REGION Network 58: Falownik P3
   // Sterowaniem pracy z falownika. Sterowanie napędem na pozycji MC
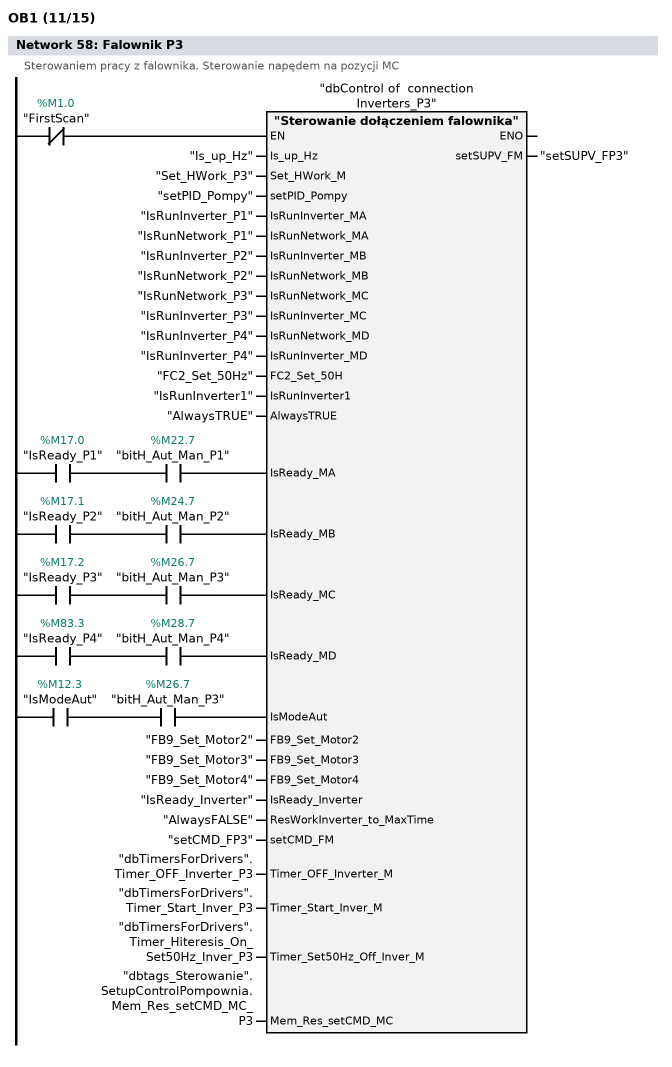
   RUNG wire#powerrail
      I_Contact( "FirstScan" )
      "dbControl of  connection Inverters_P3"(IsReady_MA := wire#w1, IsReady_MB := wire#w2, IsReady_MC := wire#w3, IsReady_MD := wire#w4, IsModeAut := wire#w5, Is_up_Hz := "Is_up_Hz", Set_HWork_M := "Set_HWork_P3", setPID_Pompy := "setPID_Pompy", IsRunInverter_MA := "IsRunInverter_P1", IsRunNetwork_MA := "IsRunNetwork_P1", IsRunInverter_MB := "IsRunInverter_P2", IsRunNetwork_MB := "IsRunNetwork_P2", IsRunNetwork_MC := "IsRunNetwork_P3", IsRunInverter_MC := "IsRunInverter_P3", IsRunNetwork_MD := "IsRunInverter_P4", IsRunInverter_MD := "IsRunInverter_P4", FC2_Set_50H := "FC2_Set_50Hz", IsRunInverter1 := "IsRunInverter1", AlwaysTRUE := "AlwaysTRUE", FB9_Set_Motor2 := "FB9_Set_Motor2", FB9_Set_Motor3 := "FB9_Set_Motor3", FB9_Set_Motor4 := "FB9_Set_Motor4", IsReady_Inverter := "IsReady_Inverter", ResWorkInverter_to_MaxTime := "AlwaysFALSE", setCMD_FM := "setCMD_FP3", Timer_OFF_Inverter_M := "dbTimersForDrivers".Timer_OFF_Inverter_P3, Timer_Start_Inver_M := "dbTimersForDrivers".Timer_Start_Inver_P3, Timer_Set50Hz_Off_Inver_M := "dbTimersForDrivers".Timer_Hiteresis_On_Set50Hz_Inver_P3, Mem_Res_setCMD_MC := "dbtags_Sterowanie".SetupControlPompownia.Mem_Res_setCMD_MC_P3, setSUPV_FM => "setSUPV_FP3")
   END_RUNG
   RUNG wire#powerrail
      Contact( "IsReady_P1" )
      Contact( "bitH_Aut_Man_P1" )
   END_RUNG wire#w1
   RUNG wire#powerrail
      Contact( "IsReady_P2" )
      Contact( "bitH_Aut_Man_P2" )
   END_RUNG wire#w2
   RUNG wire#powerrail
      Contact( "IsReady_P3" )
      Contact( "bitH_Aut_Man_P3" )
   END_RUNG wire#w3
   RUNG wire#powerrail
      Contact( "IsReady_P4" )
      Contact( "bitH_Aut_Man_P4" )
   END_RUNG wire#w4
   RUNG wire#powerrail
      Contact( "IsModeAut" )
      Contact( "bitH_Aut_Man_P3" )
   END_RUNG wire#w5
   // the same network as SCL:
   IF NOT "FirstScan" THEN
       "dbControl of  connection Inverters_P3"(Is_up_Hz := "Is_up_Hz",   // "Sterowanie dołączeniem falownika"
                               Set_HWork_M := "Set_HWork_P3",
                               setPID_Pompy := "setPID_Pompy",
                               IsRunInverter_MA := "IsRunInverter_P1",
                               IsRunNetwork_MA := "IsRunNetwork_P1",
                               IsRunInverter_MB := "IsRunInverter_P2",
                               IsRunNetwork_MB := "IsRunNetwork_P2",
                               IsRunNetwork_MC := "IsRunNetwork_P3",
                               IsRunInverter_MC := "IsRunInverter_P3",
                               IsRunNetwork_MD := "IsRunInverter_P4",
                               IsRunInverter_MD := "IsRunInverter_P4",
                               FC2_Set_50H := "FC2_Set_50Hz",
                               IsRunInverter1 := "IsRunInverter1",
                               AlwaysTRUE := "AlwaysTRUE",
                               IsReady_MA := "IsReady_P1" AND "bitH_Aut_Man_P1",
                               IsReady_MB := "IsReady_P2" AND "bitH_Aut_Man_P2",
                               IsReady_MC := "IsReady_P3" AND "bitH_Aut_Man_P3",
                               IsReady_MD := "IsReady_P4" AND "bitH_Aut_Man_P4",
                               IsModeAut := "IsModeAut" AND "bitH_Aut_Man_P3",
                               FB9_Set_Motor2 := "FB9_Set_Motor2",
                               FB9_Set_Motor3 := "FB9_Set_Motor3",
                               FB9_Set_Motor4 := "FB9_Set_Motor4",
                               IsReady_Inverter := "IsReady_Inverter",
                               ResWorkInverter_to_MaxTime := "AlwaysFALSE",
                               setCMD_FM := "setCMD_FP3",
                               Timer_OFF_Inverter_M := "dbTimersForDrivers".Timer_OFF_Inverter_P3,
                               Timer_Start_Inver_M := "dbTimersForDrivers".Timer_Start_Inver_P3,
                               Timer_Set50Hz_Off_Inver_M := "dbTimersForDrivers".Timer_Hiteresis_On_Set50Hz_Inver_P3,
                               Mem_Res_setCMD_MC := "dbtags_Sterowanie".SetupControlPompownia.Mem_Res_setCMD_MC_P3,
                               setSUPV_FM => "setSUPV_FP3");
   END_IF;
END_REGION

REGION Network 59: Falownik P4
   // Sterowaniem pracy z falownika. Sterowanie napędem na pozycji MC
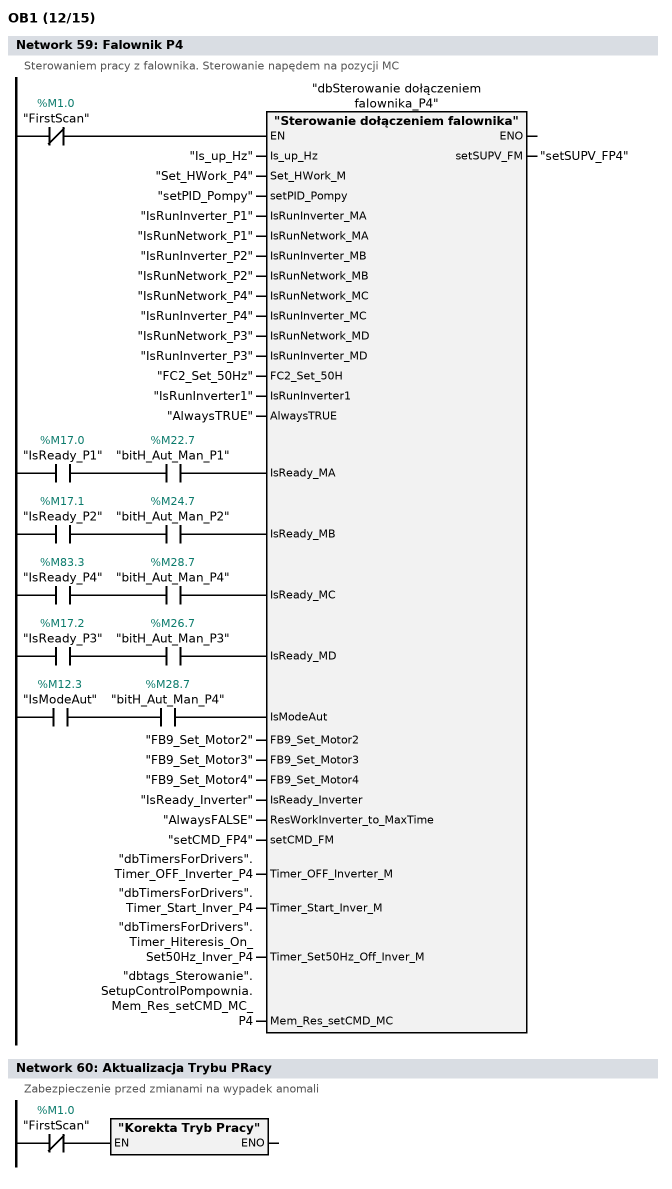
   RUNG wire#powerrail
      I_Contact( "FirstScan" )
      "dbSterowanie dołączeniem falownika_P4"(IsReady_MA := wire#w1, IsReady_MB := wire#w2, IsReady_MC := wire#w3, IsReady_MD := wire#w4, IsModeAut := wire#w5, Is_up_Hz := "Is_up_Hz", Set_HWork_M := "Set_HWork_P4", setPID_Pompy := "setPID_Pompy", IsRunInverter_MA := "IsRunInverter_P1", IsRunNetwork_MA := "IsRunNetwork_P1", IsRunInverter_MB := "IsRunInverter_P2", IsRunNetwork_MB := "IsRunNetwork_P2", IsRunNetwork_MC := "IsRunNetwork_P4", IsRunInverter_MC := "IsRunInverter_P4", IsRunNetwork_MD := "IsRunNetwork_P3", IsRunInverter_MD := "IsRunInverter_P3", FC2_Set_50H := "FC2_Set_50Hz", IsRunInverter1 := "IsRunInverter1", AlwaysTRUE := "AlwaysTRUE", FB9_Set_Motor2 := "FB9_Set_Motor2", FB9_Set_Motor3 := "FB9_Set_Motor3", FB9_Set_Motor4 := "FB9_Set_Motor4", IsReady_Inverter := "IsReady_Inverter", ResWorkInverter_to_MaxTime := "AlwaysFALSE", setCMD_FM := "setCMD_FP4", Timer_OFF_Inverter_M := "dbTimersForDrivers".Timer_OFF_Inverter_P4, Timer_Start_Inver_M := "dbTimersForDrivers".Timer_Start_Inver_P4, Timer_Set50Hz_Off_Inver_M := "dbTimersForDrivers".Timer_Hiteresis_On_Set50Hz_Inver_P4, Mem_Res_setCMD_MC := "dbtags_Sterowanie".SetupControlPompownia.Mem_Res_setCMD_MC_P4, setSUPV_FM => "setSUPV_FP4")
   END_RUNG
   RUNG wire#powerrail
      Contact( "IsReady_P1" )
      Contact( "bitH_Aut_Man_P1" )
   END_RUNG wire#w1
   RUNG wire#powerrail
      Contact( "IsReady_P2" )
      Contact( "bitH_Aut_Man_P2" )
   END_RUNG wire#w2
   RUNG wire#powerrail
      Contact( "IsReady_P4" )
      Contact( "bitH_Aut_Man_P4" )
   END_RUNG wire#w3
   RUNG wire#powerrail
      Contact( "IsReady_P3" )
      Contact( "bitH_Aut_Man_P3" )
   END_RUNG wire#w4
   RUNG wire#powerrail
      Contact( "IsModeAut" )
      Contact( "bitH_Aut_Man_P4" )
   END_RUNG wire#w5
   // the same network as SCL:
   IF NOT "FirstScan" THEN
       "dbSterowanie dołączeniem falownika_P4"(Is_up_Hz := "Is_up_Hz",   // "Sterowanie dołączeniem falownika"
                               Set_HWork_M := "Set_HWork_P4",
                               setPID_Pompy := "setPID_Pompy",
                               IsRunInverter_MA := "IsRunInverter_P1",
                               IsRunNetwork_MA := "IsRunNetwork_P1",
                               IsRunInverter_MB := "IsRunInverter_P2",
                               IsRunNetwork_MB := "IsRunNetwork_P2",
                               IsRunNetwork_MC := "IsRunNetwork_P4",
                               IsRunInverter_MC := "IsRunInverter_P4",
                               IsRunNetwork_MD := "IsRunNetwork_P3",
                               IsRunInverter_MD := "IsRunInverter_P3",
                               FC2_Set_50H := "FC2_Set_50Hz",
                               IsRunInverter1 := "IsRunInverter1",
                               AlwaysTRUE := "AlwaysTRUE",
                               IsReady_MA := "IsReady_P1" AND "bitH_Aut_Man_P1",
                               IsReady_MB := "IsReady_P2" AND "bitH_Aut_Man_P2",
                               IsReady_MC := "IsReady_P4" AND "bitH_Aut_Man_P4",
                               IsReady_MD := "IsReady_P3" AND "bitH_Aut_Man_P3",
                               IsModeAut := "IsModeAut" AND "bitH_Aut_Man_P4",
                               FB9_Set_Motor2 := "FB9_Set_Motor2",
                               FB9_Set_Motor3 := "FB9_Set_Motor3",
                               FB9_Set_Motor4 := "FB9_Set_Motor4",
                               IsReady_Inverter := "IsReady_Inverter",
                               ResWorkInverter_to_MaxTime := "AlwaysFALSE",
                               setCMD_FM := "setCMD_FP4",
                               Timer_OFF_Inverter_M := "dbTimersForDrivers".Timer_OFF_Inverter_P4,
                               Timer_Start_Inver_M := "dbTimersForDrivers".Timer_Start_Inver_P4,
                               Timer_Set50Hz_Off_Inver_M := "dbTimersForDrivers".Timer_Hiteresis_On_Set50Hz_Inver_P4,
                               Mem_Res_setCMD_MC := "dbtags_Sterowanie".SetupControlPompownia.Mem_Res_setCMD_MC_P4,
                               setSUPV_FM => "setSUPV_FP4");
   END_IF;
END_REGION

REGION Network 60: Aktualizacja Trybu PRacy
   // Zabezpieczenie przed zmianami na wypadek anomali
   RUNG wire#powerrail
      I_Contact( "FirstScan" )
      "Korekta Tryb Pracy"()
   END_RUNG
   // the same network as SCL:
   IF NOT "FirstScan" THEN "Korekta Tryb Pracy"(); END_IF;
END_REGION

REGION Network 61: Sterowanie falownikiem
   // Sterowanie załaczaniem falownika
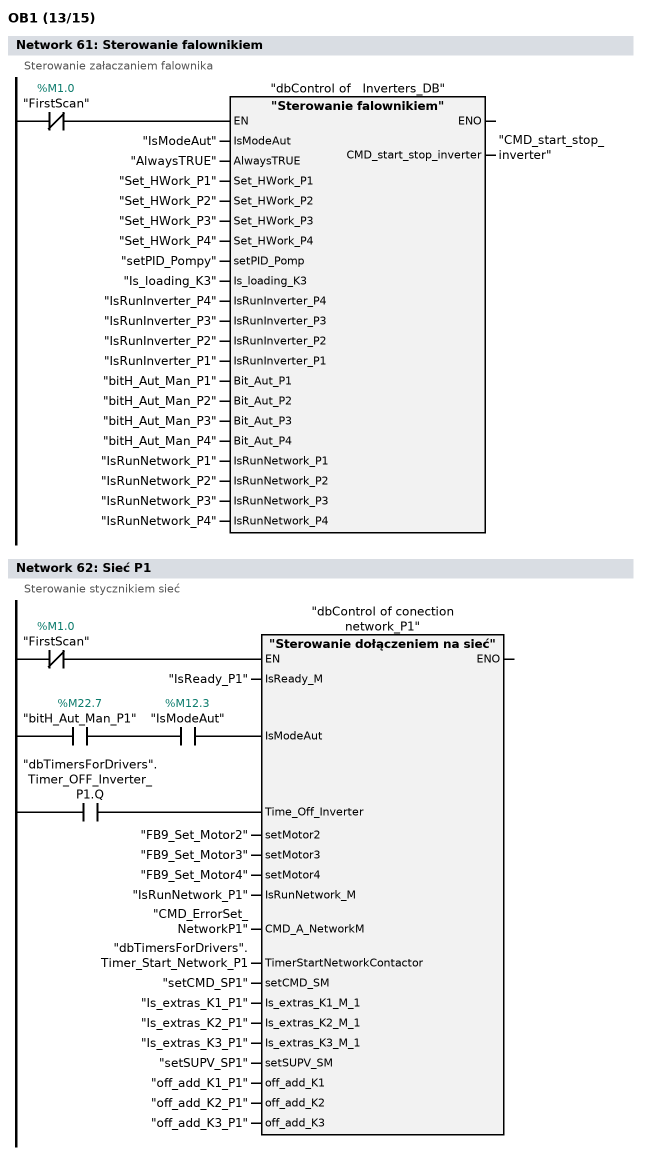
   RUNG wire#powerrail
      I_Contact( "FirstScan" )
      "dbControl of   Inverters_DB"(IsModeAut := "IsModeAut", AlwaysTRUE := "AlwaysTRUE", Set_HWork_P1 := "Set_HWork_P1", Set_HWork_P2 := "Set_HWork_P2", Set_HWork_P3 := "Set_HWork_P3", Set_HWork_P4 := "Set_HWork_P4", setPID_Pomp := "setPID_Pompy", Is_loading_K3 := "Is_loading_K3", IsRunInverter_P4 := "IsRunInverter_P4", IsRunInverter_P3 := "IsRunInverter_P3", IsRunInverter_P2 := "IsRunInverter_P2", IsRunInverter_P1 := "IsRunInverter_P1", Bit_Aut_P1 := "bitH_Aut_Man_P1", Bit_Aut_P2 := "bitH_Aut_Man_P2", Bit_Aut_P3 := "bitH_Aut_Man_P3", Bit_Aut_P4 := "bitH_Aut_Man_P4", IsRunNetwork_P1 := "IsRunNetwork_P1", IsRunNetwork_P2 := "IsRunNetwork_P2", IsRunNetwork_P3 := "IsRunNetwork_P3", IsRunNetwork_P4 := "IsRunNetwork_P4", CMD_start_stop_inverter => "CMD_start_stop_inverter")
   END_RUNG
   // the same network as SCL:
   IF NOT "FirstScan" THEN
       "dbControl of   Inverters_DB"(IsModeAut := "IsModeAut",   // "Sterowanie falownikiem"
                               AlwaysTRUE := "AlwaysTRUE",
                               Set_HWork_P1 := "Set_HWork_P1",
                               Set_HWork_P2 := "Set_HWork_P2",
                               Set_HWork_P3 := "Set_HWork_P3",
                               Set_HWork_P4 := "Set_HWork_P4",
                               setPID_Pomp := "setPID_Pompy",
                               Is_loading_K3 := "Is_loading_K3",
                               IsRunInverter_P4 := "IsRunInverter_P4",
                               IsRunInverter_P3 := "IsRunInverter_P3",
                               IsRunInverter_P2 := "IsRunInverter_P2",
                               IsRunInverter_P1 := "IsRunInverter_P1",
                               Bit_Aut_P1 := "bitH_Aut_Man_P1",
                               Bit_Aut_P2 := "bitH_Aut_Man_P2",
                               Bit_Aut_P3 := "bitH_Aut_Man_P3",
                               Bit_Aut_P4 := "bitH_Aut_Man_P4",
                               IsRunNetwork_P1 := "IsRunNetwork_P1",
                               IsRunNetwork_P2 := "IsRunNetwork_P2",
                               IsRunNetwork_P3 := "IsRunNetwork_P3",
                               IsRunNetwork_P4 := "IsRunNetwork_P4",
                               CMD_start_stop_inverter => "CMD_start_stop_inverter");
   END_IF;
END_REGION

REGION Network 62: Sieć P1
   // Sterowanie stycznikiem sieć
   RUNG wire#powerrail
      I_Contact( "FirstScan" )
      "dbControl of conection network_P1"(IsModeAut := wire#w1, Time_Off_Inverter := wire#w2, IsReady_M := "IsReady_P1", setMotor2 := "FB9_Set_Motor2", setMotor3 := "FB9_Set_Motor3", setMotor4 := "FB9_Set_Motor4", IsRunNetwork_M := "IsRunNetwork_P1", CMD_A_NetworkM := "CMD_ErrorSet_NetworkP1", TimerStartNetworkContactor := "dbTimersForDrivers".Timer_Start_Network_P1, setCMD_SM := "setCMD_SP1", Is_extras_K1_M_1 := "Is_extras_K1_P1", Is_extras_K2_M_1 := "Is_extras_K2_P1", Is_extras_K3_M_1 := "Is_extras_K3_P1", setSUPV_SM := "setSUPV_SP1", off_add_K1 := "off_add_K1_P1", off_add_K2 := "off_add_K2_P1", off_add_K3 := "off_add_K3_P1")
   END_RUNG
   RUNG wire#powerrail
      Contact( "bitH_Aut_Man_P1" )
      Contact( "IsModeAut" )
   END_RUNG wire#w1
   RUNG wire#powerrail
      Contact( "dbTimersForDrivers".Timer_OFF_Inverter_P1.Q )
   END_RUNG wire#w2
   // the same network as SCL:
   IF NOT "FirstScan" THEN
       "dbControl of conection network_P1"(IsReady_M := "IsReady_P1",   // "Sterowanie dołączeniem na sieć"
                               IsModeAut := "bitH_Aut_Man_P1" AND "IsModeAut",
                               Time_Off_Inverter := "dbTimersForDrivers".Timer_OFF_Inverter_P1.Q,
                               setMotor2 := "FB9_Set_Motor2",
                               setMotor3 := "FB9_Set_Motor3",
                               setMotor4 := "FB9_Set_Motor4",
                               IsRunNetwork_M := "IsRunNetwork_P1",
                               CMD_A_NetworkM := "CMD_ErrorSet_NetworkP1",
                               TimerStartNetworkContactor := "dbTimersForDrivers".Timer_Start_Network_P1,
                               setCMD_SM := "setCMD_SP1",
                               Is_extras_K1_M_1 := "Is_extras_K1_P1",
                               Is_extras_K2_M_1 := "Is_extras_K2_P1",
                               Is_extras_K3_M_1 := "Is_extras_K3_P1",
                               setSUPV_SM := "setSUPV_SP1",
                               off_add_K1 := "off_add_K1_P1",
                               off_add_K2 := "off_add_K2_P1",
                               off_add_K3 := "off_add_K3_P1");
   END_IF;
END_REGION

REGION Network 63: Sieć P2
   // Sterowanie stycznikiem sieć
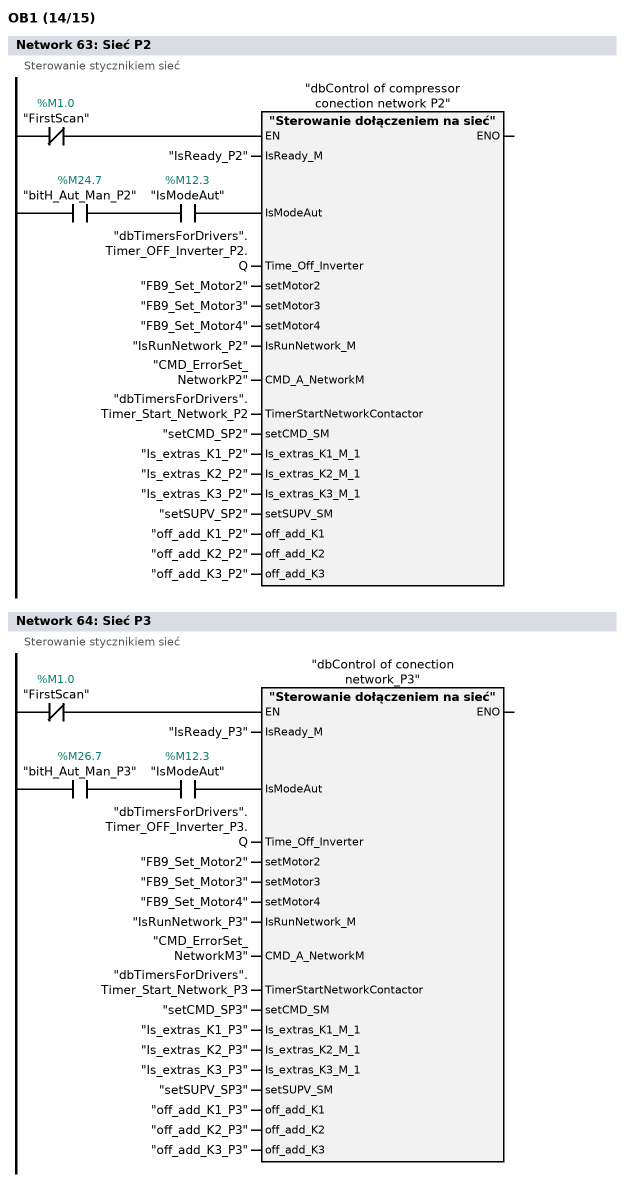
   RUNG wire#powerrail
      I_Contact( "FirstScan" )
      "dbControl of compressor conection network P2"(IsModeAut := wire#w1, IsReady_M := "IsReady_P2", Time_Off_Inverter := "dbTimersForDrivers".Timer_OFF_Inverter_P2.Q, setMotor2 := "FB9_Set_Motor2", setMotor3 := "FB9_Set_Motor3", setMotor4 := "FB9_Set_Motor4", IsRunNetwork_M := "IsRunNetwork_P2", CMD_A_NetworkM := "CMD_ErrorSet_NetworkP2", TimerStartNetworkContactor := "dbTimersForDrivers".Timer_Start_Network_P2, setCMD_SM := "setCMD_SP2", Is_extras_K1_M_1 := "Is_extras_K1_P2", Is_extras_K2_M_1 := "Is_extras_K2_P2", Is_extras_K3_M_1 := "Is_extras_K3_P2", setSUPV_SM := "setSUPV_SP2", off_add_K1 := "off_add_K1_P2", off_add_K2 := "off_add_K2_P2", off_add_K3 := "off_add_K3_P2")
   END_RUNG
   RUNG wire#powerrail
      Contact( "bitH_Aut_Man_P2" )
      Contact( "IsModeAut" )
   END_RUNG wire#w1
   // the same network as SCL:
   IF NOT "FirstScan" THEN
       "dbControl of compressor conection network P2"(IsReady_M := "IsReady_P2",   // "Sterowanie dołączeniem na sieć"
                               IsModeAut := "bitH_Aut_Man_P2" AND "IsModeAut",
                               Time_Off_Inverter := "dbTimersForDrivers".Timer_OFF_Inverter_P2.Q,
                               setMotor2 := "FB9_Set_Motor2",
                               setMotor3 := "FB9_Set_Motor3",
                               setMotor4 := "FB9_Set_Motor4",
                               IsRunNetwork_M := "IsRunNetwork_P2",
                               CMD_A_NetworkM := "CMD_ErrorSet_NetworkP2",
                               TimerStartNetworkContactor := "dbTimersForDrivers".Timer_Start_Network_P2,
                               setCMD_SM := "setCMD_SP2",
                               Is_extras_K1_M_1 := "Is_extras_K1_P2",
                               Is_extras_K2_M_1 := "Is_extras_K2_P2",
                               Is_extras_K3_M_1 := "Is_extras_K3_P2",
                               setSUPV_SM := "setSUPV_SP2",
                               off_add_K1 := "off_add_K1_P2",
                               off_add_K2 := "off_add_K2_P2",
                               off_add_K3 := "off_add_K3_P2");
   END_IF;
END_REGION

REGION Network 64: Sieć P3
   // Sterowanie stycznikiem sieć
   RUNG wire#powerrail
      I_Contact( "FirstScan" )
      "dbControl of conection network_P3"(IsModeAut := wire#w1, IsReady_M := "IsReady_P3", Time_Off_Inverter := "dbTimersForDrivers".Timer_OFF_Inverter_P3.Q, setMotor2 := "FB9_Set_Motor2", setMotor3 := "FB9_Set_Motor3", setMotor4 := "FB9_Set_Motor4", IsRunNetwork_M := "IsRunNetwork_P3", CMD_A_NetworkM := "CMD_ErrorSet_NetworkM3", TimerStartNetworkContactor := "dbTimersForDrivers".Timer_Start_Network_P3, setCMD_SM := "setCMD_SP3", Is_extras_K1_M_1 := "Is_extras_K1_P3", Is_extras_K2_M_1 := "Is_extras_K2_P3", Is_extras_K3_M_1 := "Is_extras_K3_P3", setSUPV_SM := "setSUPV_SP3", off_add_K1 := "off_add_K1_P3", off_add_K2 := "off_add_K2_P3", off_add_K3 := "off_add_K3_P3")
   END_RUNG
   RUNG wire#powerrail
      Contact( "bitH_Aut_Man_P3" )
      Contact( "IsModeAut" )
   END_RUNG wire#w1
   // the same network as SCL:
   IF NOT "FirstScan" THEN
       "dbControl of conection network_P3"(IsReady_M := "IsReady_P3",   // "Sterowanie dołączeniem na sieć"
                               IsModeAut := "bitH_Aut_Man_P3" AND "IsModeAut",
                               Time_Off_Inverter := "dbTimersForDrivers".Timer_OFF_Inverter_P3.Q,
                               setMotor2 := "FB9_Set_Motor2",
                               setMotor3 := "FB9_Set_Motor3",
                               setMotor4 := "FB9_Set_Motor4",
                               IsRunNetwork_M := "IsRunNetwork_P3",
                               CMD_A_NetworkM := "CMD_ErrorSet_NetworkM3",
                               TimerStartNetworkContactor := "dbTimersForDrivers".Timer_Start_Network_P3,
                               setCMD_SM := "setCMD_SP3",
                               Is_extras_K1_M_1 := "Is_extras_K1_P3",
                               Is_extras_K2_M_1 := "Is_extras_K2_P3",
                               Is_extras_K3_M_1 := "Is_extras_K3_P3",
                               setSUPV_SM := "setSUPV_SP3",
                               off_add_K1 := "off_add_K1_P3",
                               off_add_K2 := "off_add_K2_P3",
                               off_add_K3 := "off_add_K3_P3");
   END_IF;
END_REGION

REGION Network 65: Sieć P4
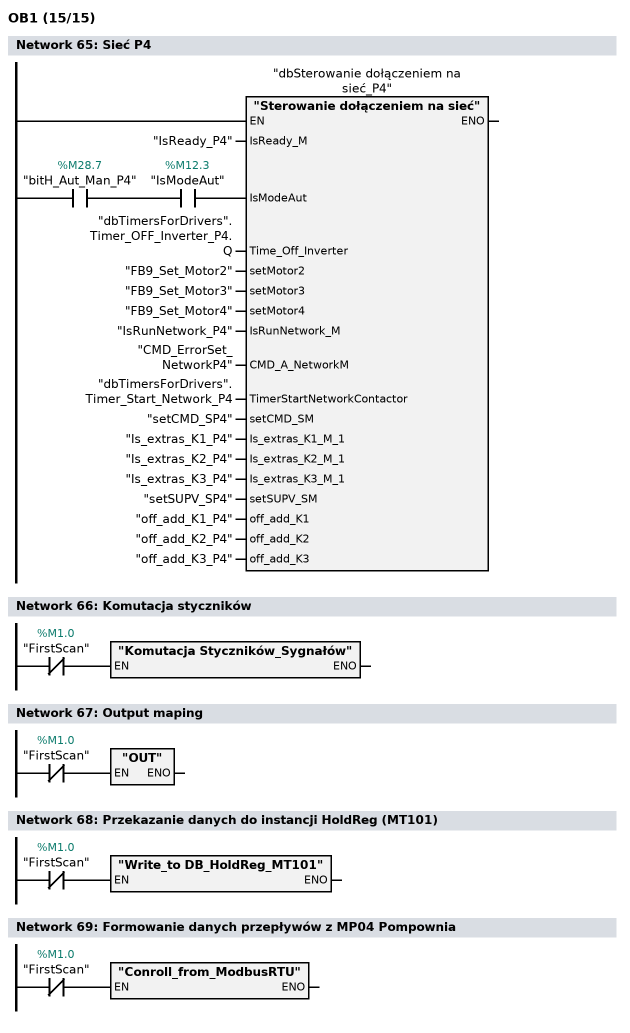
   RUNG wire#powerrail
      "dbSterowanie dołączeniem na sieć_P4"(IsModeAut := wire#w1, IsReady_M := "IsReady_P4", Time_Off_Inverter := "dbTimersForDrivers".Timer_OFF_Inverter_P4.Q, setMotor2 := "FB9_Set_Motor2", setMotor3 := "FB9_Set_Motor3", setMotor4 := "FB9_Set_Motor4", IsRunNetwork_M := "IsRunNetwork_P4", CMD_A_NetworkM := "CMD_ErrorSet_NetworkP4", TimerStartNetworkContactor := "dbTimersForDrivers".Timer_Start_Network_P4, setCMD_SM := "setCMD_SP4", Is_extras_K1_M_1 := "Is_extras_K1_P4", Is_extras_K2_M_1 := "Is_extras_K2_P4", Is_extras_K3_M_1 := "Is_extras_K3_P4", setSUPV_SM := "setSUPV_SP4", off_add_K1 := "off_add_K1_P4", off_add_K2 := "off_add_K2_P4", off_add_K3 := "off_add_K3_P4")
   END_RUNG
   RUNG wire#powerrail
      Contact( "bitH_Aut_Man_P4" )
      Contact( "IsModeAut" )
   END_RUNG wire#w1
   // the same network as SCL:
   "dbSterowanie dołączeniem na sieć_P4"(IsReady_M := "IsReady_P4",   // "Sterowanie dołączeniem na sieć"
                           IsModeAut := "bitH_Aut_Man_P4" AND "IsModeAut",
                           Time_Off_Inverter := "dbTimersForDrivers".Timer_OFF_Inverter_P4.Q,
                           setMotor2 := "FB9_Set_Motor2",
                           setMotor3 := "FB9_Set_Motor3",
                           setMotor4 := "FB9_Set_Motor4",
                           IsRunNetwork_M := "IsRunNetwork_P4",
                           CMD_A_NetworkM := "CMD_ErrorSet_NetworkP4",
                           TimerStartNetworkContactor := "dbTimersForDrivers".Timer_Start_Network_P4,
                           setCMD_SM := "setCMD_SP4",
                           Is_extras_K1_M_1 := "Is_extras_K1_P4",
                           Is_extras_K2_M_1 := "Is_extras_K2_P4",
                           Is_extras_K3_M_1 := "Is_extras_K3_P4",
                           setSUPV_SM := "setSUPV_SP4",
                           off_add_K1 := "off_add_K1_P4",
                           off_add_K2 := "off_add_K2_P4",
                           off_add_K3 := "off_add_K3_P4");
END_REGION

REGION Network 66: Komutacja styczników
   RUNG wire#powerrail
      I_Contact( "FirstScan" )
      "Komutacja Styczników_Sygnałów"()
   END_RUNG
   // the same network as SCL:
   IF NOT "FirstScan" THEN "Komutacja Styczników_Sygnałów"(); END_IF;
END_REGION

REGION Network 67: Output maping
   RUNG wire#powerrail
      I_Contact( "FirstScan" )
      "OUT"()
   END_RUNG
   // the same network as SCL:
   IF NOT "FirstScan" THEN "OUT"(); END_IF;
END_REGION

REGION Network 68: Przekazanie danych do instancji HoldReg (MT101)
   RUNG wire#powerrail
      I_Contact( "FirstScan" )
      "Write_to DB_HoldReg_MT101"()
   END_RUNG
   // the same network as SCL:
   IF NOT "FirstScan" THEN "Write_to DB_HoldReg_MT101"(); END_IF;
END_REGION

REGION Network 69: Formowanie danych przepływów z MP04 Pompownia
   RUNG wire#powerrail
      I_Contact( "FirstScan" )
      "Conroll_from_ModbusRTU"()
   END_RUNG
   // the same network as SCL:
   IF NOT "FirstScan" THEN "Conroll_from_ModbusRTU"(); END_IF;
END_REGION
END_ORGANIZATION_BLOCK

FUNCTION "RTC" : Void   // FC44, LAD
{ S7_Optimized_Access := 'TRUE' }
VERSION : 0.1
// stored: AutoNumber true, IsIECCheckEnabled false, SetENOAutomatically false, UDAEnableTagReadback false
   VAR_TEMP   // added for the SCL form of the ladder/FBD networks
      _w1 : Bool;
      _w2 : Bool;
   END_VAR
BEGIN

REGION Network 1
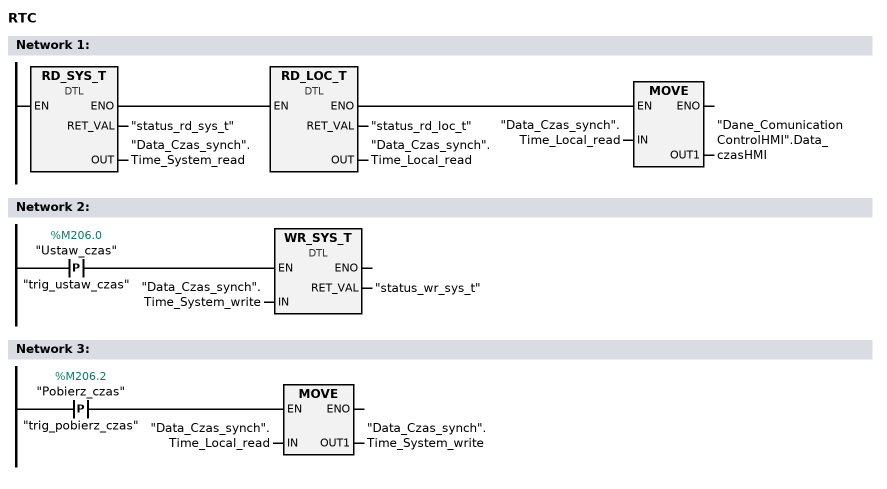
   RUNG wire#powerrail
      { S7_Templates := "date_type := DTL" } RD_SYS_T(RET_VAL => "status_rd_sys_t", OUT => "Data_Czas_synch".Time_System_read)
      { S7_Templates := "date_type := DTL" } RD_LOC_T(RET_VAL => "status_rd_loc_t", OUT => "Data_Czas_synch".Time_Local_read)
      { S7_GenerateENO := "TRUE" } Move(in := "Data_Czas_synch".Time_Local_read, out1 => "Dane_ComunicationControlHMI".Data_czasHMI)
   END_RUNG
   // the same network as SCL:
   "status_rd_sys_t" := RD_SYS_T(OUT => "Data_Czas_synch".Time_System_read, ENO => #_w1);
   "status_rd_loc_t" := RD_LOC_T(EN := #_w1, OUT => "Data_Czas_synch".Time_Local_read, ENO => #_w2);
   IF #_w2 THEN "Dane_ComunicationControlHMI".Data_czasHMI := "Data_Czas_synch".Time_Local_read; END_IF;
END_REGION

REGION Network 2
   RUNG wire#powerrail
      P_Contact(operand := "Ustaw_czas", bit := "trig_ustaw_czas")
      { S7_Templates := "date_type := DTL" } WR_SYS_T(IN := "Data_Czas_synch".Time_System_write, RET_VAL => "status_wr_sys_t")
   END_RUNG
   // the same network as SCL:
   #_w1 := "Ustaw_czas" AND NOT "trig_ustaw_czas";   // rising edge of "Ustaw_czas"
   "trig_ustaw_czas" := "Ustaw_czas";
   IF #_w1 THEN "status_wr_sys_t" := WR_SYS_T(IN := "Data_Czas_synch".Time_System_write); END_IF;
END_REGION

REGION Network 3
   RUNG wire#powerrail
      P_Contact(operand := "Pobierz_czas", bit := "trig_pobierz_czas")
      { S7_GenerateENO := "TRUE" } Move(in := "Data_Czas_synch".Time_Local_read, out1 => "Data_Czas_synch".Time_System_write)
   END_RUNG
   // the same network as SCL:
   #_w1 := "Pobierz_czas" AND NOT "trig_pobierz_czas";   // rising edge of "Pobierz_czas"
   "trig_pobierz_czas" := "Pobierz_czas";
   IF #_w1 THEN "Data_Czas_synch".Time_System_write := "Data_Czas_synch".Time_Local_read; END_IF;
END_REGION
END_FUNCTION

FUNCTION "ERR_ClassCheckError" : Void
{ S7_Optimized_Access := 'TRUE' }
VERSION : 0.1
   VAR_TEMP 
      tempCounter : Int;
   END_VAR


BEGIN
	//Get Error
	FOR #tempCounter := 0 TO 27 BY 1 DO
	    IF ("ERR_ErrorBufferFull".GetError[#tempCounter].Counter > 0) THEN
	        "V_SoftwareError".GetErrorFunction := TRUE;
	        EXIT;
	    END_IF;
	END_FOR;
	//SoftwareError   
	FOR #tempCounter := 0 TO 4 BY 1 DO
	    IF ("ERR_ErrorBufferFull".SoftwareError[#tempCounter].Counter > 0) THEN
	        "V_SoftwareError".SoftwareFunctions := TRUE;
	        EXIT;
	    END_IF;
	END_FOR;
	//OB error
	FOR #tempCounter := 0 TO 5 BY 1 DO
	    IF ("ERR_ErrorOB".OB80[#tempCounter].Counter > 0) THEN
	        "V_ErrorOB".OB80 := TRUE;
	        EXIT;
	    END_IF;
	END_FOR;
	//Diagnostic buffer
	"V_SoftwareError".DiagnosticBuffer := "ERR_ErrorBufferFull".CounterDiagStatusUpdate > 0;
	
END_FUNCTION

FUNCTION "clear_drive_error" : Void
TITLE = Modbus RTU Master do Slave przetwarzanie 
{ S7_Optimized_Access := 'TRUE' }
AUTHOR : rtecmer
VERSION : 0.1
//Funkcja przetwarz przekazane sygnały kasowania alarmów z mastera Modbus RTU (MT101) i wykonuje operację

BEGIN
	(*
	//=============================================================================
	//(JZWiK S.A Radosław Tecmer)
	//(c)Copyright (2021) All Rights Reserved
	//-----------------------------------------------------------------------------
	//Testowane z:   (system docelowy z  FW 4.2)
	//Pakiet inżynierski:   TIA Portal (V14 Sp1 Update 9)
	//Ograniczenia:  ( - )
	//Wymagania:  (minimalne S7-1200 CPU 1214 FW 3.2 .)
	//Funkcjonalnośc: (Pzetwarzanie sygnałów z MT101 protokołem Modbus RTU. 
	                    Kasowanie alarów)
	//-----------------------------------------------------------------------------
	//Zmainy wprowadzone:
	//Wersja  Data       Osoba wprowadzająca zmiany - ekspert
	//01.00.00 17.11.2021 (Tecmer Radosław - twórca) Pieresza wersja 01.00.00
	//=============================================================================
	*)
	
	//--- Kasowanie Alarmu Napędów
	
	//Ustawienie bitu Reset dla Drive Motor 1
	%DB100.DBX0.6 := %DB100.DBX51.0;
	IF %DB100.DBX1.0 = FALSE AND %DB100.DBX51.0 = TRUE  THEN
	  // ustaw automat
	  %DB100.DBX0.7 := TRUE;
	  // Kasowanie bitu RESET Driver i Modbus bit Reset
	  %DB100.DBX0.0 := FALSE;
	  %DB100.DBX51.0 := False;
	  ;
	END_IF;
	
	//Ustawienie bitu Reset dla Drive Motor 2
	%DB100.DBX2.6 := %DB100.DBX51.1;
	IF %DB100.DBX1.0 = FALSE AND %DB100.DBX51.1 =TRUE  THEN
	  // ustaw automat
	  %DB100.DBX2.7 := TRUE;
	  // Kasowanie bitu RESET Driver i Modbus bit Reset
	  %DB100.DBX2.0 := FALSE;
	  %DB100.DBX51.1 := False;
	  ;
	END_IF;
	
	//Ustawienie bitu Reset dla Drive Motor 3
	%DB100.DBX4.6 := %DB100.DBX51.2;
	IF %DB100.DBX4.0 = FALSE AND  %DB100.DBX51.2 = TRUE THEN
	  // ustaw automat
	  %DB100.DBX4.7 := TRUE;
	  // Kasowanie bitu RESET Driver i Modbus bit Reset
	  %DB100.DBX4.0 := FALSE;
	  %DB100.DBX51.2 := False;
	  ;
	END_IF;
	
	//Ustawienie bitu Reset dla Drive Motor 4
	%DB100.DBX6.6 := %DB100.DBX51.3;
	IF %DB100.DBX6.0 = FALSE AND %DB100.DBX51.3 = TRUE THEN
	  // ustaw automat
	  %DB100.DBX6.7 := TRUE;
	  // Kasowanie bitu RESET Driver i Modbus bit Reset
	  %DB100.DBX6.0 := FALSE;
	  %DB100.DBX51.3 := False;
	  ;
	END_IF;
	
	
	//Ustawienie bitu Reset dla Drive Z11
	%DB100.DBX28.6 := %DB100.DBX50.6;
	IF %DB100.DBX28.0 = FALSE AND %DB100.DBX50.6 = TRUE THEN
	  // ustaw automat
	  %DB100.DBX28.7 := TRUE;
	  // Kasowanie bitu RESET Driver i Modbus bit Reset
	  %DB100.DBX28.0 := FALSE;
	  %DB100.DBX50.6 := False;
	  ;
	END_IF;
	
	//Ustawienie bitu Reset dla Drive Z12
	%DB100.DBX30.6 := %DB100.DBX50.7;
	IF %DB100.DBX30.0 = FALSE AND %DB100.DBX50.7 =  TRUE THEN
	  // ustaw automat
	  %DB100.DBX30.7 := TRUE;
	  // Kasowanie bitu RESET Driver i Modbus bit Reset
	  %DB100.DBX30.0 := FALSE;
	  %DB100.DBX50.7 := False;
	  ;
	END_IF;
	
	// Region Zasuwy Z1 - Z10 Zbiorniki 
	//******* 
	CASE "dbHoldRegSlave_to_MT101".instClearFault1 OF
	  16:  // Ustawienie bitu Reset dla Drive Z1
	    "dbHold_RRG".Sending.rez_alarm_napędów := 16;
	    
	    ;
	  32:  // Ustawienie bitu Reset dla Drive Z2
	    "dbHold_RRG".Sending.rez_alarm_napędów := 32;
	    ;
	  64:  //Ustawienie bitu Reset dla Drive Z3
	    "dbHold_RRG".Sending.rez_alarm_napędów := 64;
	    ;
	  128:  //Ustawienie bitu Reset dla Drive Z4
	    "dbHold_RRG".Sending.rez_alarm_napędów := 128;
	    ;
	  256:  //Ustawienie bitu Reset dla Drive Z5
	    "dbHold_RRG".Sending.rez_alarm_napędów := 256;
	    ;
	  512:  //Ustawienie bitu Reset dla Drive Z6
	    "dbHold_RRG".Sending.rez_alarm_napędów := 512;
	    ;
	  1024:  //Ustawienie bitu Reset dla Drive Z7
	    "dbHold_RRG".Sending.rez_alarm_napędów := 1024;
	    ;
	  2048:  //Ustawienie bitu Reset dla Drive Z8
	    "dbHold_RRG".Sending.rez_alarm_napędów := 2048;
	    ;
	  4096:  //Ustawienie bitu Reset dla Drive Z9
	    "dbHold_RRG".Sending.rez_alarm_napędów := 4096;
	    ;
	  8192:  //Ustawienie bitu Reset dla Drive Z10
	    "dbHold_RRG".Sending.rez_alarm_napędów := 8192;
	    ;
	
	    ;
	  ELSE  // Statement section ELSE
	    ;
	END_CASE;
	
	
	// Potwierdzenie resetu alarmu Z1. Jeśli brak alarmu to wyczyść bity
	IF %DB100.DBX8.0 = FALSE  AND %DB100.DBX51.4 THEN
	  // Kasowanie bitu RESET Driver i Modbus bit Reset
	  "dbHold_RRG".Sending.rez_alarm_napędów := 0;
	  %DB100.DBX8.0 := FALSE; // bit alarm
	  %DB100.DBX51.4 := False; // bit reset
	  ;
	END_IF;
	
	// Potwierdzenie resetu alarmu Z2. Jeśli brak alarmu to wyczyść bity
	IF %DB100.DBX10.0 = FALSE AND %DB100.DBX51.5 THEN
	  // Kasowanie bitu RESET Driver i Modbus bit Reset
	  "dbHold_RRG".Sending.rez_alarm_napędów := 0;
	  %DB100.DBX10.0 := FALSE; // bit alarm
	  %DB100.DBX51.5 := False; // bit reset
	  ;
	END_IF;
	
	// Potwierdzenie resetu alarmu Z3. Jeśli brak alarmu to wyczyść bity
	IF %DB100.DBX12.0 = FALSE AND %DB100.DBX51.6 THEN
	  // Kasowanie bitu RESET Driver i Modbus bit Reset
	  "dbHold_RRG".Sending.rez_alarm_napędów := 0;
	  %DB100.DBX12.0 := FALSE; // bit alarm
	  %DB100.DBX51.6 := False; // bit reset
	  ;
	END_IF;
	
	// Potwierdzenie resetu alarmu Z4. Jeśli brak alarmu to wyczyść bity
	IF %DB100.DBX14.0 = FALSE AND %DB100.DBX51.7 THEN
	  // Kasowanie bitu RESET Driver i Modbus bit Reset
	  "dbHold_RRG".Sending.rez_alarm_napędów := 0;
	  %DB100.DBX14.0 := FALSE; // bit alarm
	  %DB100.DBX51.7 := False; // bit reset
	  ;
	END_IF;
	
	// Potwierdzenie resetu alarmu Z5. Jeśli brak alarmu to wyczyść bity
	IF %DB100.DBX16.0 = FALSE AND %DB100.DBX50.0 THEN
	  // Kasowanie bitu RESET Driver i Modbus bit Reset
	  "dbHold_RRG".Sending.rez_alarm_napędów := 0;
	  %DB100.DBX16.0 := FALSE; // bit alarm
	  %DB100.DBX50.0 := False; // bit reset
	  ;
	END_IF;
	
	// Potwierdzenie resetu alarmu Z6. Jeśli brak alarmu to wyczyść bity
	IF %DB100.DBX18.0 = FALSE AND %DB100.DBX50.1 THEN
	  // Kasowanie bitu RESET Driver i Modbus bit Reset
	  "dbHold_RRG".Sending.rez_alarm_napędów := 0;
	  %DB100.DBX18.0 := FALSE; // bit alarm
	  %DB100.DBX50.1 := False; // bit reset
	  ;
	END_IF;
	
	// Potwierdzenie resetu alarmu Z7. Jeśli brak alarmu to wyczyść bity
	IF %DB100.DBX20.0 = FALSE AND %DB100.DBX50.2 THEN
	  // Kasowanie bitu RESET Driver i Modbus bit Reset
	  "dbHold_RRG".Sending.rez_alarm_napędów := 0;
	  %DB100.DBX20.0 := FALSE; // bit alarm
	  %DB100.DBX50.2 := False; // bit reset
	  ;
	END_IF;
	
	// Potwierdzenie resetu alarmu Z8. Jeśli brak alarmu to wyczyść bity
	IF %DB100.DBX22.0 = FALSE AND %DB100.DBX50.3 THEN
	  // Kasowanie bitu RESET Driver i Modbus bit Reset
	  "dbHold_RRG".Sending.rez_alarm_napędów := 0;
	  %DB100.DBX22.0 := FALSE; // bit alarm
	  %DB100.DBX50.3 := False; // bit reset
	  ;
	END_IF;
	
	// Potwierdzenie resetu alarmu Z9. Jeśli brak alarmu to wyczyść bity
	IF %DB100.DBX24.0 = FALSE AND %DB100.DBX50.4 THEN
	  // Kasowanie bitu RESET Driver i Modbus bit Reset
	  "dbHold_RRG".Sending.rez_alarm_napędów := 0;
	  %DB100.DBX24.0 := FALSE; // bit alarm
	  %DB100.DBX50.4 := False; // bit reset
	  ;
	END_IF;
	
	// Potwierdzenie resetu alarmu Z10. Jeśli brak alarmu to wyczyść bity
	IF %DB100.DBX26.0 = FALSE AND %DB100.DBX50.5 THEN
	  // Kasowanie bitu RESET Driver i Modbus bit Reset
	  "dbHold_RRG".Sending.rez_alarm_napędów := 0;
	  %DB100.DBX26.0 := FALSE; // bit alarm
	  %DB100.DBX50.5 := False; // bit reset
	  ;
	END_IF;
	
	
	
	
	
	
	
	
	
	
	
	
END_FUNCTION

FUNCTION_BLOCK "operating_mode_select_aut-man"
TITLE = Przełącznik Trybu Pracy Napędów
{ S7_Optimized_Access := 'TRUE' }
AUTHOR : rtecmer
VERSION : 0.1
//Funkcja przeprowadza sptawdzenie stanu zmiany sygnału  na zmiennych wyboru trybu pracy napeów i jesli strwierdzi zmianę stanu zmennej to wykonuje zmianę trybu na AUT
   VAR 
      setTrig_M1 : Bool;   // bit pomocniczy przełączenia trybu
      setTrig_M2 : Bool := false;   // bit pomocniczy przełączenia trybu
      setTrig_M3 : Bool := false;   // bit pomocniczy przełączenia trybu
      setTrig_M4 : Bool := false;   // bit pomocniczy przełączenia trybu
      setTrig_Z11 : Bool := false;   // bit pomocniczy przełączenia trybu
      setTrig_Z12 : Bool := false;   // bit pomocniczy przełączenia trybu
      set_aut_man_M1 : Bool := false;   // bit pomocniczy przełączenia trybu
      set_aut_man_M2 : Bool := false;   // bit pomocniczy przełączenia trybu
      set_aut_man_M3 : Bool := false;   // bit pomocniczy przełączenia trybu
      set_aut_man_M4 : Bool := false;   // bit pomocniczy przełączenia trybu
      set_aut_man_Z11 : Bool := false;   // bit pomocniczy przełączenia trybu
      set_aut_man_Z12 : Bool := false;   // bit pomocniczy przełączenia trybu
   END_VAR


BEGIN
	(*
	//=============================================================================
	//(JZWiK S.A Radosław Tecmer)
	//(c)Copyright (2021) All Rights Reserved
	//-----------------------------------------------------------------------------
	//Testowane z:   (system docelowy z  FW 4.2)
	//Pakiet inżynierski:   TIA Portal (V14 Sp1 Update 9)
	//Ograniczenia:  ( - )
	//Wymagania:  (minimalne S7-1200 CPU 1214 FW 3.2 .)
	//Funkcjonalnośc: (Pzetwarzanie sygnałów z MT101 protokołem Modbus RTU. 
	                    Wybór Trybu Pracy Napędu)
	//-----------------------------------------------------------------------------
	//Zmainy wprowadzone:
	//Wersja  Data       Osoba wprowadzająca zmiany - ekspert
	//01.00.00 17.06.2022 (Tecmer Radosław - twórca) Pieresza wersja 01.00.00
	//=============================================================================
	*)
	
	//--- Wybór Trybu Pracy Aut/Man
	
	//Drive Motor 1 ustaw na  Automat/Manual/Start/Stop
	// Pompy
	
	REGION //Drive Motor 1 ustaw na  Automat/Manual/Start/Stop
	  // przełączniki bistabilny każdy stan Hi powoduje zmianę przełącznika
	  IF %DB100.DBX37.0 OR %DB100.DBX37.4 THEN
	    // inicjacja przełączenia
	    #set_aut_man_M1 := TRUE;
	  ELSE
	    #set_aut_man_M1 := FALSE
	    ;
	  END_IF;
	  
	  IF %DB100.DBX0.0 = FALSE THEN
	    // przełącznik bistabilny 
	    "R_TRIG_DB_AUT_M1"(CLK := #set_aut_man_M1,
	                       Q => #setTrig_M1);
	    ;
	  END_IF;
	  
	  // jeśli przełaczenie na aut
	  IF #setTrig_M1 = TRUE AND %DB100.DBX37.0 = TRUE THEN
	    %DB100.DBX0.7 := TRUE;
	    ;
	  END_IF;
	  // jeśli przełaczenie na manual
	  IF #setTrig_M1 = TRUE AND %DB100.DBX37.4 = TRUE THEN
	    %DB100.DBX0.7 := FALSE;
	    ;
	  END_IF;
	  // warunek na czyszczenie
	  IF (%DB100.DBX1.7 AND %DB100.DBX37.0) OR (%DB100.DBX1.7 = FALSE AND %DB100.DBX37.4) THEN
	    // Wyczyść całą zmienną
	    "dbHoldRegSlave_to_MT101".instConrol_ManAut_1 := 0;
	    "dbHold_Sending_TCP".Sending_Hold.set_bity_tryb_napędów_1 := 0;
	    "dbHold_RRG".Sending.set_res_bity_tryb_napędów_1 := 0;
	    // Kasowanie bitu 
	    %DB100.DBX37.0 := False;
	    %DB100.DBX37.4 := False;
	    ;
	  END_IF;
	  
	  // Start /
	  // przekazanie bitu roskazu z bloku modbus rtu do bloku statusu napędu
	IF %DB100.DBX33.0 THEN
	  // ustaw bit stat
	  %DB100.DBX0.5 := %DB100.DBX33.0; //ustawienie bitu start
	END_IF;
	IF %DB100.DBX33.0 AND %DB100.DBX0.3 THEN
	    //jeśli ustawiony bit startu z modbus i potwierdzone run napędu
	    %DB100.DBX33.0 := FALSE; // kasuj bit roskazu
	    ;
	  END_IF;
	  //Stop
	  // przekazanie bitu roskazu z bloku modbus rtu do bloku statusu napędu
	  IF %DB100.DBX33.4 THEN
	    %DB100.DBX0.4 := %DB100.DBX33.4;//ustawienie bitu stop
	    ;
	  END_IF;
	  IF %DB100.DBX33.4 AND %DB100.DBX0.3 = FALSE THEN
	    //jeśli ustawiony bit stop z modbus i potwierdzone stop napędu
	    %DB100.DBX33.4 := FALSE; // kasuj bit roskazu
	    ;
	  END_IF;
	  
	  
	  
	END_REGION
	
	
	REGION //Drive Motor 2 ustaw na  Automat/Manual/Stop/Start
	  // przełączniki bistabilny każdy stan Hi powoduje zmianę przełącznika
	  IF %DB100.DBX37.1 OR %DB100.DBX37.5 THEN
	    //inicjacja przełączenia
	    #set_aut_man_M2 := TRUE;
	  ELSE
	    #set_aut_man_M2 := FALSE
	    ;
	  END_IF;
	  
	  IF %DB100.DBX2.0 = FALSE THEN
	    // przełącznik bistabilny 
	    "R_TRIG_DB_AUT_M2"(CLK := #set_aut_man_M2,
	                       Q => #setTrig_M2);
	    ;
	  END_IF;
	  // pzrełącz na automat
	  IF #setTrig_M2 = TRUE AND %DB100.DBX37.1 = TRUE THEN
	    %DB100.DBX2.7 := TRUE;
	    ;
	  END_IF;
	  //przełącz na manual
	  IF #setTrig_M2 = TRUE AND %DB100.DBX37.5 = TRUE THEN
	    %DB100.DBX2.7 := FALSE;
	    ;
	  END_IF;
	  
	  IF (%DB100.DBX2.7 AND %DB100.DBX37.1) OR (%DB100.DBX2.7 = FALSE AND %DB100.DBX37.5)  THEN
	    // Wyczyść całą zmienną
	    "dbHoldRegSlave_to_MT101".instConrol_ManAut_1 := 0;
	    "dbHold_Sending_TCP".Sending_Hold.set_bity_tryb_napędów_1 := 0;
	    "dbHold_RRG".Sending.set_res_bity_tryb_napędów_1 := 0;
	    // Kasowanie bitu 
	    %DB100.DBX37.1 := False;
	    %DB100.DBX37.5 := FALSE;
	    ;
	  END_IF;
	  
	  // Start /
	  // przekazanie bitu roskazu z bloku modbus rtu do bloku statusu napędu
	  IF %DB100.DBX33.1 THEN // 
	    %DB100.DBX2.5 := TRUE; //ustawienie bitu start
	  END_IF;
	  IF %DB100.DBX33.1 AND %DB100.DBX2.3 THEN
	    //jeśli ustawiony bit startu z modbus i potwierdzone run napędu
	    %DB100.DBX33.1 := FALSE; // kasuj bit roskazu
	    ;
	  END_IF;
	  //Stop
	  //przekazanie bitu roskazu z bloku modbus rtu do bloku statusu napędu
	  IF %DB100.DBX33.5 THEN
	    %DB100.DBX2.4 := TRUE; //ustawienie bitu stop
	    ;
	  END_IF;
	  IF %DB100.DBX33.5 AND %DB100.DBX2.3 = FALSE THEN
	    //jeśli ustawiony bit stop z modbus i potwierdzone stop napędu
	    %DB100.DBX33.5 := FALSE; // kasuj bit roskazu
	    ;
	  END_IF;
	  
	END_REGION
	
	
	REGION //Drive Motor 3 ustaw na  Automat/Manual/Stop/Start
	  IF %DB100.DBX37.2 OR %DB100.DBX37.6 THEN
	    // przełączniki bistabilny każdy stan Hi powoduje zmianę przełącznika
	    #set_aut_man_M3 := TRUE; //ustawienie bitu start
	  ELSE
	    #set_aut_man_M3 := FALSE
	    ;
	  END_IF;
	  
	  IF %DB100.DBX4.0 = FALSE THEN
	    // przełącznik bistabilny
	    "R_TRIG_DB_AUT_M3"(CLK := #set_aut_man_M3,
	                       Q => #setTrig_M3);
	    ;
	  END_IF;
	  // przełącz na automat
	  IF #setTrig_M3 = TRUE AND %DB100.DBX37.2 = TRUE THEN
	    %DB100.DBX4.7 := TRUE;
	    ;
	  END_IF;
	  //przełącz na manual
	  IF #setTrig_M3 = TRUE AND %DB100.DBX37.6 = TRUE THEN
	    %DB100.DBX4.7 := FALSE;
	    ;
	  END_IF;
	  
	  IF (%DB100.DBX5.7 AND %DB100.DBX37.2) OR (%DB100.DBX5.7 = FALSE AND %DB100.DBX37.6) THEN
	    // Wyczyść całą zmienną
	    "dbHoldRegSlave_to_MT101".instConrol_ManAut_1 := 0;
	    "dbHold_Sending_TCP".Sending_Hold.set_bity_tryb_napędów_1 := 0;
	    "dbHold_RRG".Sending.set_res_bity_tryb_napędów_1 := 0;
	    // Kasowanie bitu 
	    %DB100.DBX37.2 := False;
	    %DB100.DBX37.6 := False;
	    ;
	  END_IF;
	  
	  // Start /
	  // przekazanie bitu roskazu z bloku modbus rtu do bloku statusu napędu
	  IF %DB100.DBX33.2 THEN
	    %DB100.DBX4.5 := TRUE; //ustawienie bitu start
	    ;
	  END_IF;
	  IF %DB100.DBX33.2 AND %DB100.DBX4.3 THEN
	    //jeśli ustawiony bit startu z modbus i potwierdzone run napędu
	    %DB100.DBX33.2 := FALSE; // kasuj bit roskazu
	    ;
	  END_IF;
	  //Stop
	  //przekazanie bitu roskazu z bloku modbus rtu do bloku statusu napędu
	  IF %DB100.DBX33.6 THEN
	    %DB100.DBX4.4 := TRUE; //ustawienie bitu stop
	    ;
	  END_IF;
	  IF %DB100.DBX33.6 AND %DB100.DBX4.3 = FALSE THEN
	    //jeśli ustawiony bit stop z modbus i potwierdzone stop napędu
	    %DB100.DBX33.6 := FALSE; // kasuj bit roskazu
	    ;
	  END_IF;
	  
	END_REGION
	
	
	REGION //Drive Motor 4 ustaw na  Automat/Manual/Stop/Start
	  IF %DB100.DBX37.3 OR %DB100.DBX37.7 THEN
	    // przełączniki bistabilny każdy stan Hi powoduje zmianę przełącznika
	    #set_aut_man_M4 := TRUE;
	  ELSE
	    #set_aut_man_M4 := FALSE
	    ;
	  END_IF;
	  
	  IF %DB100.DBX6.0 = FALSE THEN
	    // przełącznik bistabilny
	    "R_TRIG_DB_AUT_M4"(CLK := #set_aut_man_M4,
	                       Q => #setTrig_M4);
	    ;
	  END_IF;
	  
	  // przełącz na automat
	  IF #setTrig_M4 = TRUE AND %DB100.DBX37.3 = TRUE THEN
	    %DB100.DBX6.7 := TRUE;
	    ;
	  END_IF;
	  //przełącz na manual
	  IF #setTrig_M4 = TRUE AND %DB100.DBX37.7 = TRUE THEN
	    %DB100.DBX6.7 := FALSE;
	    ;
	  END_IF;
	  
	  IF (%DB100.DBX7.7 AND %DB100.DBX37.3) OR (%DB100.DBX7.7 = FALSE AND %DB100.DBX37.7) THEN
	    // Wyczyść całą zmienną
	    "dbHoldRegSlave_to_MT101".instConrol_ManAut_1 := 0;
	    "dbHold_Sending_TCP".Sending_Hold.set_bity_tryb_napędów_1 := 0;
	    "dbHold_RRG".Sending.set_res_bity_tryb_napędów_1 := 0;
	    // Kasowanie bitu 
	    %DB100.DBX37.3 := False;
	    %DB100.DBX37.7:= FALSE
	    ;
	  END_IF;
	  
	  // Start /
	  // przekazanie bitu roskazu z bloku modbus rtu do bloku statusu napędu
	  IF %DB100.DBX33.3 THEN
	    %DB100.DBX6.5 := TRUE; //ustawienie bitu start
	    ;
	  END_IF;
	  IF %DB100.DBX33.3 AND %DB100.DBX6.3 THEN
	    //jeśli ustawiony bit startu z modbus i potwierdzone run napędu
	    %DB100.DBX33.3 := FALSE; // kasuj bit roskazu
	    ;
	  END_IF;
	  //Stop
	  //przekazanie bitu roskazu z bloku modbus rtu do bloku statusu napędu
	  IF %DB100.DBX33.7 THEN
	    %DB100.DBX6.4 := TRUE; //ustawienie bitu stop
	    ;
	  END_IF;
	  IF %DB100.DBX33.7 AND %DB100.DBX6.3 = FALSE THEN
	    //jeśli ustawiony bit stop z modbus i potwierdzone stop napędu
	    %DB100.DBX33.7 := FALSE; // kasuj bit roskazu
	    ;
	  END_IF;
	  
	  
	END_REGION
	
	// Zasuwy
	
	REGION //Drive Motor Z11 ustaw na  Automat/Manual/Otwieranie/Zamykanie
	  IF %DB100.DBX39.2 OR %DB100.DBX38.6 THEN
	    // przełączniki bistabilny każdy stan Hi powoduje zmianę przełącznika
	    #set_aut_man_Z11 := TRUE;
	  ELSE
	    #set_aut_man_Z11 := FALSE
	    ;
	  END_IF;
	  
	  IF %DB100.DBX28.0 = FALSE THEN
	    // przełącznik bistabilny
	    "R_TRIG_DB_AUT_Z11"(CLK := #set_aut_man_Z11,
	                        Q => #setTrig_Z11);
	    ;
	  END_IF;
	  //przełącz na automay
	  IF #setTrig_Z11 = TRUE AND %DB100.DBX39.2 = TRUE THEN
	    %DB100.DBX28.7 := TRUE;
	    ;
	  END_IF;
	  //przełącz na manual
	  IF #setTrig_Z11 = TRUE AND %DB100.DBX38.6 = TRUE THEN
	    %DB100.DBX28.7 := FALSE;
	    ;
	  END_IF;
	  
	  IF (%DB100.DBX29.7 AND %DB100.DBX39.2) OR (%DB100.DBX29.7 = FALSE AND %DB100.DBX38.6) THEN
	    // Wyczyść całą zmienną
	    "dbHoldRegSlave_to_MT101".instConrol_ManAut_2 := 0;
	    "dbHold_Sending_TCP".Sending_Hold.set_bity_tryb_napędów_2 := 0;
	    "dbHold_RRG".Sending.set_res_bity_tryb_napędów_2 := 0;
	    // Kasowanie bitu 
	    %DB100.DBX39.2 := False;
	    %DB100.DBX38.6 := FALSE
	    ;
	  END_IF;
	  
	  // Otwórz/
	  // przekazanie bitu roskazu z bloku modbus rtu do bloku statusu napędu
	  IF %DB100.DBX35.2 THEN
	    %DB100.DBX28.4 := %DB100.DBX35.2; //ustawienie bitu otwieranie
	    ;
	  END_IF;
	  IF %DB100.DBX35.2 AND %DB100.DBX29.1 THEN
	    //jeśli ustawiony bit otwierania z modbus i potwierdzone otwarcie 
	    %DB100.DBX35.2 := FALSE; // kasuj bit roskazu
	    ;
	  END_IF;
	  //Zamknij
	  //przekazanie bitu roskazu z bloku modbus rtu do bloku statusu napędu
	  IF %DB100.DBX34.6 THEN
	    %DB100.DBX28.5 := %DB100.DBX34.6; //ustawienie bitu zamykanie
	    ;
	  END_IF;
	  IF %DB100.DBX34.6 AND %DB100.DBX29.3 = FALSE THEN
	    //jeśli ustawiony bit zamykaniez modbus i potwierdzone zamknięcie 
	    %DB100.DBX34.6 := FALSE; // kasuj bit roskazu
	    ;
	  END_IF;
	  
	END_REGION
	
	
	REGION //Drive Motor Z12 ustaw na  Automat/Manual/Otwieranie/Zamykanie
	  IF %DB100.DBX39.3 OR %DB100.DBX38.7 THEN
	    // przełączniki bistabilny każdy stan Hi powoduje zmianę przełącznika
	    #set_aut_man_Z12 := TRUE;
	  ELSE
	    #set_aut_man_Z12 := FALSE
	    ;
	  END_IF;
	  
	  IF %DB100.DBX30.0 = FALSE THEN
	    // przełącznik bistabilny
	    "R_TRIG_DB_AUT_Z12"(CLK := #set_aut_man_Z12,
	                        Q => #setTrig_Z12);
	    ;
	  END_IF;
	  // przełącz na automat
	  IF #setTrig_Z12 = TRUE AND %DB100.DBX39.3 = TRUE THEN
	    %DB100.DBX30.7 := TRUE;
	    ;
	  END_IF;
	  // przełącz na manual
	  IF #setTrig_Z12 = TRUE AND %DB100.DBX38.7 = TRUE THEN
	    %DB100.DBX30.7 := FALSE;
	    ;
	  END_IF;
	  
	  IF (%DB100.DBX31.7 AND %DB100.DBX39.3) OR (%DB100.DBX31.7 = FALSE AND %DB100.DBX38.7) THEN
	    // Wyczyść całą zmienną
	    "dbHoldRegSlave_to_MT101".instConrol_ManAut_2 := 0;
	    "dbHold_Sending_TCP".Sending_Hold.set_bity_tryb_napędów_2 := 0;
	    "dbHold_RRG".Sending.set_res_bity_tryb_napędów_2 := 0;
	    // Kasowanie bitu 
	    %DB100.DBX39.3 := FALSE;
	    %DB100.DBX38.7:= FALSE
	    ;
	  END_IF;
	  
	  // Otwórz/
	  // przekazanie bitu roskazu z bloku modbus rtu do bloku statusu napędu
	  IF %DB100.DBX35.3 THEN
	    %DB100.DBX30.4 := %DB100.DBX35.3; //ustawienie bitu otwieranie
	    ;
	  END_IF;
	  IF %DB100.DBX35.3 AND %DB100.DBX31.1 THEN
	    //jeśli ustawiony bit otwierania z modbus i potwierdzone otwarcie 
	    %DB100.DBX35.3 := FALSE; // kasuj bit roskazu
	    ;
	  END_IF;
	  //Zamknij
	  //przekazanie bitu roskazu z bloku modbus rtu do bloku statusu napędu
	  IF %DB100.DBX34.7 THEN
	    %DB100.DBX30.5 := %DB100.DBX34.7; //ustawienie bitu zamykanie
	    ;
	  END_IF;
	  %DB100.DBX30.5 := %DB100.DBX34.7; //ustawienie bitu zamykanie
	  IF %DB100.DBX34.7 AND %DB100.DBX31.3 = FALSE THEN
	    //jeśli ustawiony bit zamykaniez modbus i potwierdzone zamknięcie 
	    %DB100.DBX34.7 := FALSE; // kasuj bit roskazu
	    ;
	  END_IF;
	  
	END_REGION
	
	
	(* 
	 ------------------------------------------------------------------------
	 
	Część obsługi PLC-2 obsługa czyszczenia zmiennych po odebraniu potwierdzeń  
	---------------------------------------------------------------------------
	*)
	
	REGION //Drive Motor Z1 ustaw na  Automat/Manual
	  //sprawdzenie czy wyłano polecenie przełaczenia w Aut i czy bit Aut napędu jest True
	  IF ("dbHold_Sending_TCP".Sending_Hold.set_bity_tryb_napędów_1 = 256 AND %DB100.DBX8.7)
	    OR
	    //sprawdzenie czy wyłano polecenie przełaczenia w Man i czy bit Aut napędu jest False
	    ("dbHold_Sending_TCP".Sending_Hold.set_bity_tryb_napędów_2 = 16 AND %DB100.DBX8.7 = FALSE)
	  THEN
	    // Jeśli któryś z warunków spełniony wyczyść 
	    "dbHold_Sending_TCP".Sending_Hold.set_bity_tryb_napędów_1 := 0;
	    "dbHold_RRG".Sending.set_res_bity_tryb_napędów_1 := 0;
	    "dbHold_Sending_TCP".Sending_Hold.set_bity_tryb_napędów_2 := 0;
	    "dbHold_RRG".Sending.set_res_bity_tryb_napędów_2 := 0;
	    
	  END_IF;
	  
	  //  przesyłanie rozkazów OTWIERANIE - ZAMYKANIE
	  //------------OTWIERANIE - ZAMYKANIE
	  //sprawdzenie czy wyłano polecenie otwieranie i czy bit otwieranie jest True
	  IF ("dbHold_Sending_TCP".Sending_Hold.set_bity_sterowania_napęami_1 = 256 AND %DB100.DBX8.1)
	    OR
	    //sprawdzenie czy wyłano polecenie zamykanie i czy bit zamykanie jest true
	    ("dbHold_Sending_TCP".Sending_Hold.set_bity_sterowania_napęami_2 = 16 AND %DB100.DBX8.3)
	  THEN
	    // Jeśli któryś z warunków spełniony wyczyść 
	    "dbHold_Sending_TCP".Sending_Hold.set_bity_sterowania_napęami_1 := 0;
	    "dbHold_RRG".Sending.set_res_bity_sterowania_napęami_1 := 0;
	    "dbHold_Sending_TCP".Sending_Hold.set_bity_sterowania_napęami_2 := 0;
	    "dbHold_RRG".Sending.set_res_bity_sterowania_napęami_2 := 0;
	  END_IF;
	  
	  
	END_REGION
	
	REGION //Drive Motor Z2 ustaw na  Automat/Manual
	  IF ("dbHold_Sending_TCP".Sending_Hold.set_bity_tryb_napędów_1 = 512 AND %DB100.DBX10.7)
	    OR
	    ("dbHold_Sending_TCP".Sending_Hold.set_bity_tryb_napędów_2 = 32 AND %DB100.DBX10.7 = FALSE)
	  THEN
	    // Wyczyść całą zmienną
	    "dbHold_Sending_TCP".Sending_Hold.set_bity_tryb_napędów_1 := 0;
	    "dbHold_RRG".Sending.set_res_bity_tryb_napędów_1 := 0;
	    "dbHold_Sending_TCP".Sending_Hold.set_bity_tryb_napędów_2 := 0;
	    "dbHold_RRG".Sending.set_res_bity_tryb_napędów_2 := 0;
	    ;
	  END_IF;
	  
	    //  przesyłanie rozkazów OTWIERANIE - ZAMYKANIE
	  //------------OTWIERANIE - ZAMYKANIE
	  //sprawdzenie czy wyłano polecenie otwieranie i czy bit otwieranie jest True
	  IF ("dbHold_Sending_TCP".Sending_Hold.set_bity_sterowania_napęami_1 = 512 AND %DB100.DBX10.1)
	    OR
	    //sprawdzenie czy wyłano polecenie zamykanie i czy bit zamykanie jest true
	    ("dbHold_Sending_TCP".Sending_Hold.set_bity_sterowania_napęami_2 = 32 AND %DB100.DBX10.3)
	  THEN
	    // Jeśli któryś z warunków spełniony wyczyść 
	    "dbHold_Sending_TCP".Sending_Hold.set_bity_sterowania_napęami_1 := 0;
	    "dbHold_RRG".Sending.set_res_bity_sterowania_napęami_1 := 0;
	    "dbHold_Sending_TCP".Sending_Hold.set_bity_sterowania_napęami_2 := 0;
	    "dbHold_RRG".Sending.set_res_bity_sterowania_napęami_2 := 0;
	  END_IF;
	  
	END_REGION
	
	REGION //Drive Motor Z3 ustaw na  Automat/Manual
	  IF ("dbHold_Sending_TCP".Sending_Hold.set_bity_tryb_napędów_1 = 1024 AND %DB100.DBX12.7)
	    OR
	    ("dbHold_Sending_TCP".Sending_Hold.set_bity_tryb_napędów_2 = 64 AND %DB100.DBX12.7 = FALSE)
	  THEN
	    // Wyczyść całą zmienną
	    "dbHold_Sending_TCP".Sending_Hold.set_bity_tryb_napędów_1 := 0;
	    "dbHold_RRG".Sending.set_res_bity_tryb_napędów_1 := 0;
	    "dbHold_Sending_TCP".Sending_Hold.set_bity_tryb_napędów_2 := 0;
	    "dbHold_RRG".Sending.set_res_bity_tryb_napędów_2 := 0;
	    ;
	  END_IF;
	  
	  //  przesyłanie rozkazów OTWIERANIE - ZAMYKANIE
	  //------------OTWIERANIE - ZAMYKANIE
	  //sprawdzenie czy wyłano polecenie otwieranie i czy bit otwieranie jest True
	  IF ("dbHold_Sending_TCP".Sending_Hold.set_bity_sterowania_napęami_1 = 1024 AND %DB100.DBX12.1)
	    OR
	    //sprawdzenie czy wyłano polecenie zamykanie i czy bit zamykanie jest true
	    ("dbHold_Sending_TCP".Sending_Hold.set_bity_sterowania_napęami_2 = 64 AND %DB100.DBX12.3)
	  THEN
	    // Jeśli któryś z warunków spełniony wyczyść 
	    "dbHold_Sending_TCP".Sending_Hold.set_bity_sterowania_napęami_1 := 0;
	    "dbHold_RRG".Sending.set_res_bity_sterowania_napęami_1 := 0;
	    "dbHold_Sending_TCP".Sending_Hold.set_bity_sterowania_napęami_2 := 0;
	    "dbHold_RRG".Sending.set_res_bity_sterowania_napęami_2 := 0;
	  END_IF;
	  
	END_REGION
	
	REGION //Drive Motor Z4 ustaw na  Automat/Manual
	  IF ("dbHold_Sending_TCP".Sending_Hold.set_bity_tryb_napędów_1 = 2048 AND %DB100.DBX14.7)
	    OR
	    ("dbHold_Sending_TCP".Sending_Hold.set_bity_tryb_napędów_2 = 128 AND %DB100.DBX14.7 = FALSE)
	  THEN
	    // Wyczyść całą zmienną
	    "dbHold_Sending_TCP".Sending_Hold.set_bity_tryb_napędów_1 := 0;
	    "dbHold_RRG".Sending.set_res_bity_tryb_napędów_1 := 0;
	    "dbHold_Sending_TCP".Sending_Hold.set_bity_tryb_napędów_2 := 0;
	    "dbHold_RRG".Sending.set_res_bity_tryb_napędów_2 := 0;
	    ;
	  END_IF;
	  
	  //  przesyłanie rozkazów OTWIERANIE - ZAMYKANIE
	  //------------OTWIERANIE - ZAMYKANIE
	  //sprawdzenie czy wyłano polecenie otwieranie i czy bit otwieranie jest True
	  IF ("dbHold_Sending_TCP".Sending_Hold.set_bity_sterowania_napęami_1 = 2048 AND %DB100.DBX14.1)
	    OR
	    //sprawdzenie czy wyłano polecenie zamykanie i czy bit zamykanie jest true
	    ("dbHold_Sending_TCP".Sending_Hold.set_bity_sterowania_napęami_2 = 128 AND %DB100.DBX14.3)
	  THEN
	    // Jeśli któryś z warunków spełniony wyczyść 
	    "dbHold_Sending_TCP".Sending_Hold.set_bity_sterowania_napęami_1 := 0;
	    "dbHold_RRG".Sending.set_res_bity_sterowania_napęami_1 := 0;
	    "dbHold_Sending_TCP".Sending_Hold.set_bity_sterowania_napęami_2 := 0;
	    "dbHold_RRG".Sending.set_res_bity_sterowania_napęami_2 := 0;
	  END_IF;
	  
	END_REGION
	
	REGION //Drive Motor Z5 ustaw na Automat/Manual
	  IF ("dbHold_Sending_TCP".Sending_Hold.set_bity_tryb_napędów_1 = 4096 AND %DB100.DBX16.7)
	    OR
	    ("dbHold_Sending_TCP".Sending_Hold.set_bity_tryb_napędów_2 = 256 AND %DB100.DBX16.7 = FALSE)
	  THEN
	    // Wyczyść całą zmienną
	    "dbHold_Sending_TCP".Sending_Hold.set_bity_tryb_napędów_1 := 0;
	    "dbHold_RRG".Sending.set_res_bity_tryb_napędów_1 := 0;
	    "dbHold_Sending_TCP".Sending_Hold.set_bity_tryb_napędów_2 := 0;
	    "dbHold_RRG".Sending.set_res_bity_tryb_napędów_2 := 0;
	    ;
	  END_IF;
	  
	  //  przesyłanie rozkazów OTWIERANIE - ZAMYKANIE
	  //------------OTWIERANIE - ZAMYKANIE
	  //sprawdzenie czy wyłano polecenie otwieranie i czy bit otwieranie jest True
	  IF ("dbHold_Sending_TCP".Sending_Hold.set_bity_sterowania_napęami_1 = 4096 AND %DB100.DBX16.1)
	    OR
	    //sprawdzenie czy wyłano polecenie zamykanie i czy bit zamykanie jest true
	    ("dbHold_Sending_TCP".Sending_Hold.set_bity_sterowania_napęami_2 = 256 AND %DB100.DBX16.3)
	  THEN
	    // Jeśli któryś z warunków spełniony wyczyść 
	    "dbHold_Sending_TCP".Sending_Hold.set_bity_sterowania_napęami_1 := 0;
	    "dbHold_RRG".Sending.set_res_bity_sterowania_napęami_1 := 0;
	    "dbHold_Sending_TCP".Sending_Hold.set_bity_sterowania_napęami_2 := 0;
	    "dbHold_RRG".Sending.set_res_bity_sterowania_napęami_2 := 0;
	  END_IF;
	  
	END_REGION
	
	REGION //Drive Motor Z6 ustaw na  Automat/Manual
	  IF ("dbHold_Sending_TCP".Sending_Hold.set_bity_tryb_napędów_1 = 8192 AND %DB100.DBX18.7)
	    OR
	    ("dbHold_Sending_TCP".Sending_Hold.set_bity_tryb_napędów_2 = 512 AND %DB100.DBX18.7 = FALSE)
	  THEN
	    // Wyczyść całą zmienną
	    "dbHold_Sending_TCP".Sending_Hold.set_bity_tryb_napędów_1 := 0;
	    "dbHold_RRG".Sending.set_res_bity_tryb_napędów_1 := 0;
	    "dbHold_Sending_TCP".Sending_Hold.set_bity_tryb_napędów_2 := 0;
	    "dbHold_RRG".Sending.set_res_bity_tryb_napędów_2 := 0;
	    ;
	  END_IF;
	  
	  //  przesyłanie rozkazów OTWIERANIE - ZAMYKANIE
	  //------------OTWIERANIE - ZAMYKANIE
	  //sprawdzenie czy wyłano polecenie otwieranie i czy bit otwieranie jest True
	  IF ("dbHold_Sending_TCP".Sending_Hold.set_bity_sterowania_napęami_1 = 8192 AND %DB100.DBX18.1)
	    OR
	    //sprawdzenie czy wyłano polecenie zamykanie i czy bit zamykanie jest true
	    ("dbHold_Sending_TCP".Sending_Hold.set_bity_sterowania_napęami_2 = 512 AND %DB100.DBX18.3)
	  THEN
	    // Jeśli któryś z warunków spełniony wyczyść 
	    "dbHold_Sending_TCP".Sending_Hold.set_bity_sterowania_napęami_1 := 0;
	    "dbHold_RRG".Sending.set_res_bity_sterowania_napęami_1 := 0;
	    "dbHold_Sending_TCP".Sending_Hold.set_bity_sterowania_napęami_2 := 0;
	    "dbHold_RRG".Sending.set_res_bity_sterowania_napęami_2 := 0;
	  END_IF;
	  
	END_REGION
	
	REGION //Drive Motor Z7 ustaw na  Automat/Manual
	  IF ("dbHold_Sending_TCP".Sending_Hold.set_bity_tryb_napędów_1 = 16384 AND %DB100.DBX20.7)
	    OR
	    ("dbHold_Sending_TCP".Sending_Hold.set_bity_tryb_napędów_2 = 1024 AND %DB100.DBX20.7 = FALSE)
	  THEN
	    // Wyczyść całą zmienną
	    "dbHold_Sending_TCP".Sending_Hold.set_bity_tryb_napędów_1 := 0;
	    "dbHold_RRG".Sending.set_res_bity_tryb_napędów_1 := 0;
	    "dbHold_Sending_TCP".Sending_Hold.set_bity_tryb_napędów_2 := 0;
	    "dbHold_RRG".Sending.set_res_bity_tryb_napędów_2 := 0;
	    ;
	  END_IF;
	  
	  //  przesyłanie rozkazów OTWIERANIE - ZAMYKANIE
	  //------------OTWIERANIE - ZAMYKANIE
	  //sprawdzenie czy wyłano polecenie otwieranie i czy bit otwieranie jest True
	  IF ("dbHold_Sending_TCP".Sending_Hold.set_bity_sterowania_napęami_1 = 16384 AND %DB100.DBX20.1)
	    
	    OR
	    //sprawdzenie czy wyłano polecenie zamykanie i czy bit zamykanie jest true
	    ("dbHold_Sending_TCP".Sending_Hold.set_bity_sterowania_napęami_2 = 1024 AND %DB100.DBX20.3)
	  THEN
	    // Jeśli któryś z warunków spełniony wyczyść 
	    "dbHold_Sending_TCP".Sending_Hold.set_bity_sterowania_napęami_1 := 0;
	    "dbHold_RRG".Sending.set_res_bity_sterowania_napęami_1 := 0;
	    "dbHold_Sending_TCP".Sending_Hold.set_bity_sterowania_napęami_2 := 0;
	    "dbHold_RRG".Sending.set_res_bity_sterowania_napęami_2 := 0;
	  END_IF;
	  
	END_REGION
	
	REGION //Drive Motor Z8 ustaw na Automat/Manual
	  IF ("dbHold_Sending_TCP".Sending_Hold.set_bity_tryb_napędów_1 = 32768 AND %DB100.DBX22.7)
	    OR
	    ("dbHold_Sending_TCP".Sending_Hold.set_bity_tryb_napędów_2 = 2048 AND %DB100.DBX22.7 = FALSE)
	  THEN
	    // Wyczyść całą zmienną
	    "dbHold_Sending_TCP".Sending_Hold.set_bity_tryb_napędów_1 := 0;
	    "dbHold_RRG".Sending.set_res_bity_tryb_napędów_1 := 0;
	    "dbHold_Sending_TCP".Sending_Hold.set_bity_tryb_napędów_2 := 0;
	    "dbHold_RRG".Sending.set_res_bity_tryb_napędów_2 := 0;
	    ;
	  END_IF;
	  
	  //  przesyłanie rozkazów OTWIERANIE - ZAMYKANIE
	  //------------OTWIERANIE - ZAMYKANIE
	  //sprawdzenie czy wyłano polecenie otwieranie i czy bit otwieranie jest True
	  IF ("dbHold_Sending_TCP".Sending_Hold.set_bity_sterowania_napęami_1 = 32768 AND %DB100.DBX22.1)
	    OR
	    //sprawdzenie czy wyłano polecenie zamykanie i czy bit zamykanie jest true
	    ("dbHold_Sending_TCP".Sending_Hold.set_bity_sterowania_napęami_2 = 2048 AND %DB100.DBX22.3)
	  THEN
	    // Jeśli któryś z warunków spełniony wyczyść 
	    "dbHold_Sending_TCP".Sending_Hold.set_bity_sterowania_napęami_1 := 0;
	    "dbHold_RRG".Sending.set_res_bity_sterowania_napęami_1 := 0;
	    "dbHold_Sending_TCP".Sending_Hold.set_bity_sterowania_napęami_2 := 0;
	    "dbHold_RRG".Sending.set_res_bity_sterowania_napęami_2 := 0;
	  END_IF;
	  
	END_REGION
	
	REGION //Drive Motor Z9 ustaw na  Automat/Manual
	  IF ("dbHold_Sending_TCP".Sending_Hold.set_bity_tryb_napędów_2 = 1 AND %DB100.DBX24.7)
	    OR
	    ("dbHold_Sending_TCP".Sending_Hold.set_bity_tryb_napędów_2 = 4096 AND %DB100.DBX24.7 = FALSE)
	  THEN
	    // Wyczyść całą zmienną
	    "dbHold_Sending_TCP".Sending_Hold.set_bity_tryb_napędów_2 := 0;
	    "dbHold_RRG".Sending.set_res_bity_tryb_napędów_2 := 0;
	    ;
	  END_IF;
	  
	  //  przesyłanie rozkazów OTWIERANIE - ZAMYKANIE
	  //------------OTWIERANIE - ZAMYKANIE
	  //sprawdzenie czy wyłano polecenie otwieranie i czy bit otwieranie jest True
	  IF ("dbHold_Sending_TCP".Sending_Hold.set_bity_sterowania_napęami_2 = 1 AND %DB100.DBX24.1)
	    OR
	    //sprawdzenie czy wyłano polecenie zamykanie i czy bit zamykanie jest true
	    ("dbHold_Sending_TCP".Sending_Hold.set_bity_sterowania_napęami_2 = 4096 AND %DB100.DBX24.3)
	  THEN
	    // Jeśli któryś z warunków spełniony wyczyść 
	    "dbHold_Sending_TCP".Sending_Hold.set_bity_sterowania_napęami_2 := 0;
	    "dbHold_RRG".Sending.set_res_bity_sterowania_napęami_2 := 0;
	    "dbHold_Sending_TCP".Sending_Hold.set_bity_sterowania_napęami_1 := 0;
	    "dbHold_RRG".Sending.set_res_bity_sterowania_napęami_1 := 0;
	  END_IF;
	  
	
	  
	END_REGION
	
	REGION //Drive Motor Z10 ustaw na  Automat/Manual
	  IF ("dbHold_Sending_TCP".Sending_Hold.set_bity_tryb_napędów_2 = 2 AND %DB100.DBX26.7)
	    OR
	    ("dbHold_Sending_TCP".Sending_Hold.set_bity_tryb_napędów_2 = 8192 AND %DB100.DBX26.7 = FALSE)
	  THEN
	    // Wyczyść całą zmienną
	    "dbHold_Sending_TCP".Sending_Hold.set_bity_tryb_napędów_2 := 0;
	    "dbHold_RRG".Sending.set_res_bity_tryb_napędów_2 := 0;
	    ;
	  END_IF;
	  
	  //  przesyłanie rozkazów OTWIERANIE - ZAMYKANIE
	  //------------OTWIERANIE - ZAMYKANIE
	  //sprawdzenie czy wyłano polecenie otwieranie i czy bit otwieranie jest True
	  IF ("dbHold_Sending_TCP".Sending_Hold.set_bity_sterowania_napęami_2 = 2 AND %DB100.DBX26.1)
	    OR
	    //sprawdzenie czy wyłano polecenie zamykanie i czy bit zamykanie jest true
	    ("dbHold_Sending_TCP".Sending_Hold.set_bity_sterowania_napęami_2 = 8192 AND %DB100.DBX26.3)
	  THEN
	    // Jeśli któryś z warunków spełniony wyczyść 
	    "dbHold_Sending_TCP".Sending_Hold.set_bity_sterowania_napęami_2 := 0;
	    "dbHold_RRG".Sending.set_res_bity_sterowania_napęami_2 := 0;
	    "dbHold_Sending_TCP".Sending_Hold.set_bity_sterowania_napęami_1 := 0;
	    "dbHold_RRG".Sending.set_res_bity_sterowania_napęami_1 := 0;
	  END_IF;
	  
	END_REGION
	
	
	
	
	
	
	
	
	
	
	
	
	
	
	
	
	
	
	
	  
	
	
	
	
END_FUNCTION_BLOCK

FUNCTION "ParsowanieDataTime_Zadanych_" : Void
TITLE = Persowanie danych data i time
{ S7_Optimized_Access := 'TRUE' }
AUTHOR : rtecmer
VERSION : 0.1
//Funkcja składa z wartości podanego czasu formie Real zmienne DTL przekazywane dale do układu sterowania zbiornikami i pompami

BEGIN
	(*
	//=============================================================================
	//(JZWiK S.A Radosław Tecmer)
	//(c)Copyright (2022) All Rights Reserved
	//-----------------------------------------------------------------------------
	//Testowane z:   (system docelowy z  FW 4.4)
	//Pakiet inżynierski:   TIA Portal (V16 Update 5)
	//Ograniczenia:  ( - )
	//Wymagania:  (minimalne S7-1200 CPU 1215C FW 4.2 .)
	//Funkcjonalnośc: (Persowanie danych wchodzących w formie Real do danych DTL
	                    Dane: czasy, sterowania zbiornikami i pracą pomp)
	//-----------------------------------------------------------------------------
	//Zmainy wprowadzone:
	//Wersja  Data       Osoba wprowadzająca zmiany - ekspert
	//01.00.00 09.03.2022 (Tecmer Radosław - twórca) Pieresza wersja 01.00.00
	//=============================================================================
	*)
	
	
	REGION start_napełnianie
	  // przekazanie z bloku SCADA do bloku danych programu PLC
	  "db10organizacyjna".instHourStart_Filling.HOUR := INT_TO_USINT("dbHoldRegSlave_to_MT101".instHourStart_Filling);
	  "db10organizacyjna".instHourStart_Filling.MINUTE := INT_TO_USINT("dbHoldRegSlave_to_MT101".instMinutStart_Filling);
	  "dbHold_RRG".SendingTimes.start_napełnianie.SECOND := 0;
	  // przekazanie do bloku danych wysyłanych 
	  "dbHold_RRG".SendingTimes.start_napełnianie.YEAR := "Data_Czas_synch".Time_Local_read.YEAR;
	  "dbHold_RRG".SendingTimes.start_napełnianie.MONTH := "Data_Czas_synch".Time_Local_read.MONTH;
	  "dbHold_RRG".SendingTimes.start_napełnianie.DAY := "Data_Czas_synch".Time_Local_read.DAY;
	  "dbHold_RRG".SendingTimes.start_napełnianie.WEEKDAY := "Data_Czas_synch".Time_Local_read.WEEKDAY;
	  //"dbHold_RRG".SendingTimes.start_napełnianie.HOUR := INT_TO_USINT("dbHoldRegSlave_to_MT101".Godziny.instHourStart_Filling);
	  //"dbHold_RRG".SendingTimes.start_napełnianie.MINUTE := INT_TO_USINT("dbHoldRegSlave_to_MT101".Godziny.instMinutStart_Filling);
	  "dbHold_RRG".SendingTimes.start_napełnianie.SECOND := 0;
	  
	END_REGION
	
	REGION Stop_napełnianie
	  // przekazanie z bloku SCADA do bloku danych programu PLC
	  "db10organizacyjna".instHourStop_Filling.HOUR := INT_TO_USINT("dbHoldRegSlave_to_MT101".instHourStop_Filling);
	  "db10organizacyjna".instHourStop_Filling.MINUTE := INT_TO_USINT("dbHoldRegSlave_to_MT101".instMinutStopt_Filling);
	  "dbHold_RRG".SendingTimes.Stop_napełnianie.SECOND := 0;
	  // przekazanie do bloku danych wysyłanych 
	  "dbHold_RRG".SendingTimes.Stop_napełnianie.YEAR := "Data_Czas_synch".Time_Local_read.YEAR;
	  "dbHold_RRG".SendingTimes.Stop_napełnianie.MONTH := "Data_Czas_synch".Time_Local_read.MONTH;
	  "dbHold_RRG".SendingTimes.Stop_napełnianie.DAY := "Data_Czas_synch".Time_Local_read.DAY;
	  "dbHold_RRG".SendingTimes.Stop_napełnianie.WEEKDAY := "Data_Czas_synch".Time_Local_read.WEEKDAY;
	  //"dbHold_RRG".SendingTimes.Stop_napełnianie.HOUR := INT_TO_USINT("dbHoldRegSlave_to_MT101".Godziny.instHourStop_Filling);
	  //"dbHold_RRG".SendingTimes.Stop_napełnianie.MINUTE := INT_TO_USINT("dbHoldRegSlave_to_MT101".Godziny.instMinutStopt_Filling);
	  "dbHold_RRG".SendingTimes.Stop_napełnianie.SECOND := 0;
	  
	END_REGION
	
	REGION Start_przetłaczanie_1
	  //
	  "db10organizacyjna".instHourStart_City.HOUR := INT_TO_USINT("dbHoldRegSlave_to_MT101".instHourStart_City);
	  "db10organizacyjna".instHourStart_City.MINUTE := INT_TO_USINT("dbHoldRegSlave_to_MT101".instMinutStart_City);
	  "dbHold_RRG".SendingTimes.Start_przetłaczanie_1.SECOND := 0;
	  //  przekazanie do bloku danych wysyłanych 
	  "dbHold_RRG".SendingTimes.Start_przetłaczanie_1.YEAR := "Data_Czas_synch".Time_Local_read.YEAR;
	  "dbHold_RRG".SendingTimes.Start_przetłaczanie_1.MONTH := "Data_Czas_synch".Time_Local_read.MONTH;
	  "dbHold_RRG".SendingTimes.Start_przetłaczanie_1.DAY := "Data_Czas_synch".Time_Local_read.DAY;
	  "dbHold_RRG".SendingTimes.Start_przetłaczanie_1.WEEKDAY := "Data_Czas_synch".Time_Local_read.WEEKDAY;
	  //"dbHold_RRG".SendingTimes.Start_przetłaczanie_1.HOUR := INT_TO_USINT("dbHoldRegSlave_to_MT101".Godziny.instHourStart_City);
	 // "dbHold_RRG".SendingTimes.Start_przetłaczanie_1.MINUTE := INT_TO_USINT("dbHoldRegSlave_to_MT101".Godziny.instMinutStart_City);
	  "dbHold_RRG".SendingTimes.Start_przetłaczanie_1.SECOND := 0;
	  
	END_REGION
	
	REGION Stop_przetłaczanie_1
	  // przekazanie z bloku SCADA do bloku danych programu PLC
	  "db10organizacyjna".instHourStop_City.HOUR := INT_TO_USINT("dbHoldRegSlave_to_MT101".instHourStop_City);
	  "db10organizacyjna".instHourStop_City.MINUTE := INT_TO_USINT("dbHoldRegSlave_to_MT101".instMinutStopt_City);
	  "dbHold_RRG".SendingTimes.Stop_przetłaczanie_1.SECOND := 0;
	  // przekazanie do bloku danych wysyłanych 
	  "dbHold_RRG".SendingTimes.Stop_przetłaczanie_1.YEAR := "Data_Czas_synch".Time_Local_read.YEAR;
	  "dbHold_RRG".SendingTimes.Stop_przetłaczanie_1.MONTH := "Data_Czas_synch".Time_Local_read.MONTH;
	  "dbHold_RRG".SendingTimes.Stop_przetłaczanie_1.DAY := "Data_Czas_synch".Time_Local_read.DAY;
	  "dbHold_RRG".SendingTimes.Stop_przetłaczanie_1.WEEKDAY := "Data_Czas_synch".Time_Local_read.WEEKDAY;
	 // "dbHold_RRG".SendingTimes.Stop_przetłaczanie_1.HOUR := INT_TO_USINT("dbHoldRegSlave_to_MT101".Godziny.instHourStop_City);
	 // "dbHold_RRG".SendingTimes.Stop_przetłaczanie_1.MINUTE := INT_TO_USINT("dbHoldRegSlave_to_MT101".Godziny.instMinutStopt_City);
	  "dbHold_RRG".SendingTimes.Stop_przetłaczanie_1.SECOND := 0;
	  
	END_REGION
	
	REGION Start_dosilanie_1
	  // przekazanie z bloku SCADA do bloku danych programu PLC
	  "db10organizacyjna".instHourStart_Replen.HOUR := INT_TO_USINT("dbHoldRegSlave_to_MT101".instHourStart_Replen);
	  "db10organizacyjna".instHourStart_Replen.MINUTE := INT_TO_USINT("dbHoldRegSlave_to_MT101".instMinutStart_Replen);
	  "dbHold_RRG".SendingTimes.Start_dosilanie_1.SECOND := 0;
	  // przekazanie do bloku danych wysyłanych 
	  "dbHold_RRG".SendingTimes.Start_dosilanie_1.YEAR := "Data_Czas_synch".Time_Local_read.YEAR;
	  "dbHold_RRG".SendingTimes.Start_dosilanie_1.MONTH := "Data_Czas_synch".Time_Local_read.MONTH;
	  "dbHold_RRG".SendingTimes.Start_dosilanie_1.DAY := "Data_Czas_synch".Time_Local_read.DAY;
	  "dbHold_RRG".SendingTimes.Start_dosilanie_1.WEEKDAY := "Data_Czas_synch".Time_Local_read.WEEKDAY;
	  //"dbHold_RRG".SendingTimes.Start_dosilanie_1.HOUR := INT_TO_USINT("dbHoldRegSlave_to_MT101".Godziny.instHourStart_Replen);
	  //"dbHold_RRG".SendingTimes.Start_dosilanie_1.MINUTE := INT_TO_USINT("dbHoldRegSlave_to_MT101".Godziny.instMinutStart_Replen);
	  "dbHold_RRG".SendingTimes.Start_dosilanie_1.SECOND := 0;
	  
	END_REGION
	
	REGION Stop_dosilanie_1
	  // przekazanie z bloku SCADA do bloku danych programu PLC
	  "db10organizacyjna".instHourStop_Replen.HOUR := INT_TO_USINT("dbHoldRegSlave_to_MT101".instHourStop_Replen);
	  "db10organizacyjna".instHourStop_Replen.MINUTE := INT_TO_USINT("dbHoldRegSlave_to_MT101".instMinutStopt_Replen);
	  "dbHold_RRG".SendingTimes.Stop_dosilanie_1.SECOND := 0;
	  // przekazanie do bloku danych wysyłanych 
	  "dbHold_RRG".SendingTimes.Stop_dosilanie_1.YEAR := "Data_Czas_synch".Time_Local_read.YEAR;
	  "dbHold_RRG".SendingTimes.Stop_dosilanie_1.MONTH := "Data_Czas_synch".Time_Local_read.MONTH;
	  "dbHold_RRG".SendingTimes.Stop_dosilanie_1.DAY := "Data_Czas_synch".Time_Local_read.DAY;
	  "dbHold_RRG".SendingTimes.Stop_dosilanie_1.WEEKDAY := "Data_Czas_synch".Time_Local_read.WEEKDAY;
	  //"dbHold_RRG".SendingTimes.Stop_dosilanie_1.HOUR := INT_TO_USINT("dbHoldRegSlave_to_MT101".Godziny.instHourStop_Replen);
	  //"dbHold_RRG".SendingTimes.Stop_dosilanie_1.MINUTE := INT_TO_USINT("dbHoldRegSlave_to_MT101".Godziny.instMinutStopt_Replen);
	  "dbHold_RRG".SendingTimes.Stop_dosilanie_1.SECOND := 0;
	END_REGION
	
	
	
	
	
	
	
	
	
	
	
	
	
	
END_FUNCTION

FUNCTION "Czyszczenie_błednych_wpisów" : Void
TITLE = Korekta błednego wpisu
{ S7_Optimized_Access := 'TRUE' }
AUTHOR : rtecmer
VERSION : 0.1
//Program kontroluje błedny wpis wartości poza granicą liczby określającej czas (godziny, minuty) W razie wpisania złej wartości wypełna komurkę zerami

BEGIN
	(*
	//=============================================================================
	//(JZWiK S.A Radosław Tecmer)
	//(c)Copyright (2022) All Rights Reserved
	//-----------------------------------------------------------------------------
	//Testowane z:   (system docelowy z  FW 4.4)
	//Pakiet inżynierski:   TIA Portal (V16 Update 5)
	//Ograniczenia:  ( - )
	//Wymagania:  (minimalne S7-1200 CPU 1215C FW 4.2 .)
	//Funkcjonalnośc: (Kontrola błednego wpisy wartości liczbowej czasu, wartości.
	                   Jeśli wartość poza zakresem wypełnieni komórki zerami)
	//-----------------------------------------------------------------------------
	//Zmainy wprowadzone:
	//Wersja  Data       Osoba wprowadzająca zmiany - ekspert
	//01.00.00 05.05.2022 (Tecmer Radosław - twórca) Pieresza wersja 01.00.00
	//=============================================================================
	*)
	
	
	
	
	
	//poziomy
	
	//napełnianie
	IF "dbHoldRegSlave_to_MT101".instLevelSetFilling < 0
	  OR "dbHoldRegSlave_to_MT101".instLevelSetFilling > 1000
	  OR "dbHold_RRG".Sending.set_poziom_napełniania < 0
	  OR "dbHold_RRG".Sending.set_poziom_napełniania > 1000
	THEN
	  // wypełnij zerami
	  "dbHoldRegSlave_to_MT101".instLevelSetFilling := 0;
	  "dbHold_Sending_TCP".Sending_Hold.set_poziom_napełniania := 0;
	  "dbHold_RRG".set_poziom_napełniania := 0;
	  ;
	END_IF;
	
	//opróżnianie
	IF "dbHoldRegSlave_to_MT101".instLevelSetEmptying < 0
	  OR "dbHoldRegSlave_to_MT101".instLevelSetEmptying > 1000
	  OR "dbHold_RRG".Sending.set_poziom_opróżniania < 0
	  OR "dbHold_RRG".Sending.set_poziom_opróżniania > 1000
	  OR "dbHoldRegSlave_to_MT101".instLevelSetEmptying >= "dbHoldRegSlave_to_MT101".instLevelSetFilling
	  OR "dbHold_RRG".Sending.set_poziom_opróżniania >= "dbHold_RRG".Sending.set_poziom_napełniania
	THEN
	  // wypełnij zerami
	  "dbHoldRegSlave_to_MT101".instLevelSetEmptying := 0;
	  "dbHold_Sending_TCP".Sending_Hold.set_poziom_opróżniania := 0;
	  "dbHold_RRG".Sending.set_poziom_opróżniania := 0;
	  ;
	END_IF;
	
	
	// zadane położenie zasuwy Z10
	IF "dbHoldRegSlave_to_MT101".instPosition_Z10 < 0
	  OR "dbHoldRegSlave_to_MT101".instPosition_Z10 > 100
	  OR "dbHold_RRG".Sending.set_położenie_Z10 < 0
	  OR "dbHold_RRG".Sending.set_położenie_Z10 > 100
	THEN
	  // wypełnij zerami
	  "dbHoldRegSlave_to_MT101".instPosition_Z10 := 0;
	  "dbHold_Sending_TCP".Sending_Hold.set_położenie_Z10 := 0;
	  "dbHold_RRG".Sending.set_położenie_Z10 := 0; 
	  
	END_IF;
	
	
	// czasy
	// 
	// napełnianie on
	IF "dbHoldRegSlave_to_MT101".instHourStart_Filling < 0
	  OR "dbHoldRegSlave_to_MT101".instHourStart_Filling > 23
	  OR "dbHold_Sending_TCP".Sending_Hold.instHourStart_Filling <0
	  OR "dbHold_Sending_TCP".Sending_Hold.instHourStart_Filling > 23
	THEN
	  // wypełnij zerami
	  "dbHoldRegSlave_to_MT101".instHourStart_Filling := 0;
	  "dbHold_Sending_TCP".Sending_Hold.instHourStart_Filling:= 0;
	  "dbHold_RRG".start_napełnianie.HOUR := 0;
	  ;
	END_IF;
	
	IF "dbHoldRegSlave_to_MT101".instMinutStart_Filling < 0
	  OR "dbHoldRegSlave_to_MT101".instMinutStart_Filling > 60
	    OR "dbHold_RRG".SendingTimes.start_napełnianie.MINUTE < 0
	    OR "dbHold_RRG".SendingTimes.start_napełnianie.MINUTE > 60
	  THEN
	    // wypełnij zerami
	    "dbHoldRegSlave_to_MT101".instMinutStart_Filling := 0;
	    "dbHold_Sending_TCP".Sending_Hold.instMinutStart_Filling := 0;
	    "dbHold_RRG".start_napełnianie.MINUTE := 0;
	    "dbHold_RRG".SendingTimes.start_napełnianie.MINUTE := 0;
	    ;
	END_IF;
	
	// napełnianie off
	IF "dbHoldRegSlave_to_MT101".instHourStop_Filling < 0
	  OR "dbHoldRegSlave_to_MT101".instHourStop_Filling > 23
	  OR "dbHold_RRG".SendingTimes.Stop_napełnianie.HOUR < 0
	  OR "dbHold_RRG".SendingTimes.Stop_napełnianie.HOUR > 23
	THEN
	  // wypełnij zerami
	  "dbHoldRegSlave_to_MT101".instHourStop_Filling := 0;
	  "dbHold_Sending_TCP".Sending_Hold.instHourStop_Filling := 0;
	  "dbHold_RRG".SendingTimes.Stop_napełnianie.HOUR := 0;
	  ;
	END_IF;
	
	IF "dbHoldRegSlave_to_MT101".instMinutStopt_Filling < 0
	  OR "dbHoldRegSlave_to_MT101".instMinutStopt_Filling > 60
	  OR "dbHold_RRG".SendingTimes.Stop_napełnianie.MINUTE < 0
	  OR "dbHold_RRG".SendingTimes.Stop_napełnianie.MINUTE > 60
	THEN
	  // wypełnij zerami
	  "dbHoldRegSlave_to_MT101".instMinutStopt_Filling := 0;
	  "dbHold_Sending_TCP".Sending_Hold.instMinutStopt_Filling := 0;
	  "dbHold_RRG".SendingTimes.Stop_napełnianie.MINUTE := 0;
	  ;
	END_IF;
	
	
	// przetłaczanie on
	IF "dbHoldRegSlave_to_MT101".instHourStart_City < 0
	  OR "dbHoldRegSlave_to_MT101".instHourStart_City > 23
	  OR "dbHold_RRG".SendingTimes.Start_przetłaczanie_1.HOUR < 0
	  OR "dbHold_RRG".SendingTimes.Start_przetłaczanie_1.HOUR > 23
	THEN
	  // wypełnij zerami
	  "dbHoldRegSlave_to_MT101".instHourStart_City := 0;
	  "dbHold_Sending_TCP".Sending_Hold.instHourStart_City := 0;
	  "dbHold_RRG".SendingTimes.Start_przetłaczanie_1.HOUR := 0;
	  ;
	END_IF;
	
	IF "dbHoldRegSlave_to_MT101".instMinutStart_City < 0
	  OR "dbHoldRegSlave_to_MT101".instMinutStart_City > 60
	  OR "dbHold_RRG".SendingTimes.Start_przetłaczanie_1.MINUTE < 0
	  OR "dbHold_RRG".SendingTimes.Start_przetłaczanie_1.MINUTE > 60
	THEN
	  // wypełnij zerami
	  "dbHoldRegSlave_to_MT101".instMinutStart_City := 0;
	  "dbHold_Sending_TCP".Sending_Hold.instMinutStart_City := 0;
	  "dbHold_RRG".SendingTimes.Start_przetłaczanie_1.MINUTE := 0;
	  ;
	END_IF;
	
	// przetłaczanie off
	IF "dbHoldRegSlave_to_MT101".instHourStop_City < 0
	  OR "dbHoldRegSlave_to_MT101".instHourStop_City > 23
	  OR "dbHold_RRG".SendingTimes.Stop_przetłaczanie_1.HOUR < 0
	  OR "dbHold_RRG".SendingTimes.Stop_przetłaczanie_1.HOUR > 23
	THEN
	  // wypełnij zerami
	  "dbHoldRegSlave_to_MT101".instHourStop_City := 0;
	  "dbHold_Sending_TCP".Sending_Hold.instHourStop_City := 0;
	  "dbHold_RRG".SendingTimes.Stop_przetłaczanie_1.HOUR := 0;
	  ;
	END_IF;
	
	IF "dbHoldRegSlave_to_MT101".instMinutStopt_City < 0
	  OR "dbHoldRegSlave_to_MT101".instMinutStopt_City > 60
	  OR "dbHold_RRG".SendingTimes.Stop_przetłaczanie_1.MINUTE < 0
	  OR "dbHold_RRG".SendingTimes.Stop_przetłaczanie_1.MINUTE > 60
	THEN
	  // wypełnij zerami
	  "dbHoldRegSlave_to_MT101".instMinutStopt_City := 0;
	  "dbHold_Sending_TCP".Sending_Hold.instMinutStopt_City := 0;
	  "dbHold_RRG".SendingTimes.Stop_przetłaczanie_1.MINUTE := 0;
	  ;
	END_IF;
	
	//dosilanie on
	IF "dbHoldRegSlave_to_MT101".instHourStart_Replen < 0
	  OR "dbHoldRegSlave_to_MT101".instHourStart_Replen > 23
	  OR "dbHold_RRG".SendingTimes.Start_dosilanie_1.HOUR < 0
	  OR "dbHold_RRG".SendingTimes.Start_dosilanie_1.HOUR > 23
	THEN
	  // wypełnij zerami
	  "dbHoldRegSlave_to_MT101".instHourStart_Replen := 0;
	  "dbHold_Sending_TCP".Sending_Hold.instHourStart_Replen := 0;
	  "dbHold_RRG".SendingTimes.Start_dosilanie_1.HOUR := 0;
	  ;
	END_IF;
	
	IF "dbHoldRegSlave_to_MT101".instMinutStart_Replen < 0
	  OR "dbHoldRegSlave_to_MT101".instMinutStart_Replen > 60
	  OR "dbHold_RRG".SendingTimes.Start_dosilanie_1.MINUTE < 0
	  OR "dbHold_RRG".SendingTimes.Start_dosilanie_1.MINUTE > 60
	THEN
	  // wypełnij zerami
	  "dbHoldRegSlave_to_MT101".instMinutStart_Replen := 0;
	  "dbHold_Sending_TCP".Sending_Hold.instMinutStart_Replen := 0;
	  "dbHold_RRG".SendingTimes.Start_dosilanie_1.MINUTE := 0;
	  ;
	END_IF;
	
	//dosilanie off
	IF "dbHoldRegSlave_to_MT101".instHourStop_Replen < 0
	  OR "dbHoldRegSlave_to_MT101".instHourStop_Replen > 23
	  OR "dbHold_RRG".SendingTimes.Stop_dosilanie_1.HOUR < 0
	  OR "dbHold_RRG".SendingTimes.Stop_dosilanie_1.HOUR  > 23
	THEN
	  // wypełnij zerami
	  "dbHoldRegSlave_to_MT101".instHourStop_Replen := 0;
	  "dbHold_Sending_TCP".Sending_Hold.instHourStop_Replen := 0;
	  "dbHold_RRG".SendingTimes.Stop_dosilanie_1.HOUR := 0;
	  ;
	END_IF;
	
	IF "dbHoldRegSlave_to_MT101".instMinutStopt_Replen < 0
	  OR "dbHoldRegSlave_to_MT101".instMinutStopt_Replen > 60
	  OR "dbHold_RRG".SendingTimes.Stop_dosilanie_1.MINUTE < 0
	  OR "dbHold_RRG".SendingTimes.Stop_dosilanie_1.MINUTE > 60
	THEN
	  // wypełnij zerami
	  "dbHoldRegSlave_to_MT101".instMinutStopt_Replen := 0;
	  "dbHold_Sending_TCP".Sending_Hold.instMinutStopt_Replen := 0;
	  "dbHold_RRG".SendingTimes.Stop_dosilanie_1.MINUTE := 0;
	  ;
	END_IF;
	
	
	
	
	
	
END_FUNCTION

FUNCTION_BLOCK "Modbus_TCP"   // FB6, LAD
TITLE = Wywołanie funkcji MB_Server
{ S7_Optimized_Access := 'TRUE' }
AUTHOR : rtecmer
VERSION : 0.1
// stored: AutoNumber true, IsIECCheckEnabled false, IsRetainMemResEnabled false, MemoryReserve 100, SetENOAutomatically false, UDAEnableTagReadback false
   VAR_TEMP   // added for the SCL form of the ladder/FBD networks
      _w1 : Bool;
   END_VAR
BEGIN

REGION Network 1: Sewrer
   // Wpisywane z PLC 2 Zbiorniki
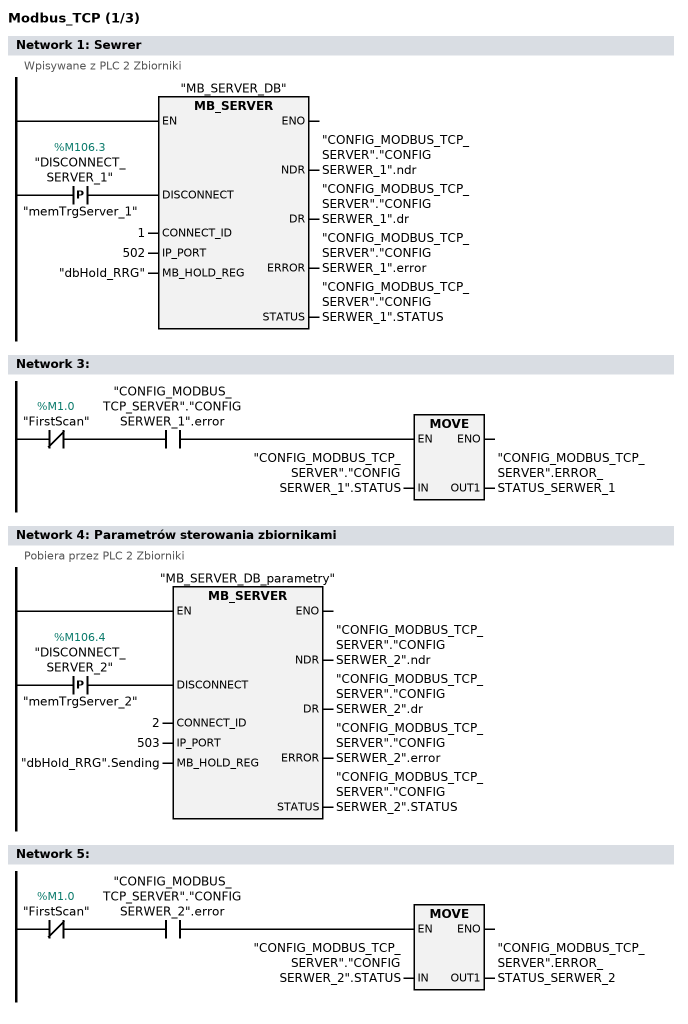
   RUNG wire#powerrail
      { S7_Templates := "[card1200 := 1, card1500 := 0]" } "MB_SERVER_DB".MB_SERVER(DISCONNECT := wire#w1, CONNECT_ID := 1, IP_PORT := 502, MB_HOLD_REG := "dbHold_RRG", NDR => "CONFIG_MODBUS_TCP_SERVER"."CONFIG SERWER_1".ndr, DR => "CONFIG_MODBUS_TCP_SERVER"."CONFIG SERWER_1".dr, ERROR => "CONFIG_MODBUS_TCP_SERVER"."CONFIG SERWER_1".error, STATUS => "CONFIG_MODBUS_TCP_SERVER"."CONFIG SERWER_1".STATUS)
   END_RUNG
   RUNG wire#powerrail
      P_Contact(operand := "DISCONNECT_SERVER_1", bit := "memTrgServer_1")
   END_RUNG wire#w1
   // the same network as SCL:
   #_w1 := "DISCONNECT_SERVER_1" AND NOT "memTrgServer_1";   // rising edge of "DISCONNECT_SERVER_1"
   "memTrgServer_1" := "DISCONNECT_SERVER_1";
   "MB_SERVER_DB"(DISCONNECT := #_w1,   // MB_SERVER
                  CONNECT_ID := 1,
                  IP_PORT := 502,
                  MB_HOLD_REG := "dbHold_RRG",
                  NDR => "CONFIG_MODBUS_TCP_SERVER"."CONFIG SERWER_1".ndr,
                  DR => "CONFIG_MODBUS_TCP_SERVER"."CONFIG SERWER_1".dr,
                  ERROR => "CONFIG_MODBUS_TCP_SERVER"."CONFIG SERWER_1".error,
                  STATUS => "CONFIG_MODBUS_TCP_SERVER"."CONFIG SERWER_1".STATUS);
END_REGION

REGION Network 3
   RUNG wire#powerrail
      I_Contact( "FirstScan" )
      Contact( "CONFIG_MODBUS_TCP_SERVER"."CONFIG SERWER_1".error )
      Move(in := "CONFIG_MODBUS_TCP_SERVER"."CONFIG SERWER_1".STATUS, out1 => "CONFIG_MODBUS_TCP_SERVER".ERROR_STATUS_SERWER_1)
   END_RUNG
   // the same network as SCL:
   IF NOT "FirstScan" AND "CONFIG_MODBUS_TCP_SERVER"."CONFIG SERWER_1".error THEN
       "CONFIG_MODBUS_TCP_SERVER".ERROR_STATUS_SERWER_1 := "CONFIG_MODBUS_TCP_SERVER"."CONFIG SERWER_1".STATUS;
   END_IF;
END_REGION

REGION Network 4: Parametrów sterowania zbiornikami
   // Pobiera przez PLC 2 Zbiorniki
   RUNG wire#powerrail
      { S7_Templates := "[card1200 := 1, card1500 := 0]" } "MB_SERVER_DB_parametry".MB_SERVER(DISCONNECT := wire#w1, CONNECT_ID := 2, IP_PORT := 503, MB_HOLD_REG := "dbHold_RRG".Sending, NDR => "CONFIG_MODBUS_TCP_SERVER"."CONFIG SERWER_2".ndr, DR => "CONFIG_MODBUS_TCP_SERVER"."CONFIG SERWER_2".dr, ERROR => "CONFIG_MODBUS_TCP_SERVER"."CONFIG SERWER_2".error, STATUS => "CONFIG_MODBUS_TCP_SERVER"."CONFIG SERWER_2".STATUS)
   END_RUNG
   RUNG wire#powerrail
      P_Contact(operand := "DISCONNECT_SERVER_2", bit := "memTrgServer_2")
   END_RUNG wire#w1
   // the same network as SCL:
   #_w1 := "DISCONNECT_SERVER_2" AND NOT "memTrgServer_2";   // rising edge of "DISCONNECT_SERVER_2"
   "memTrgServer_2" := "DISCONNECT_SERVER_2";
   "MB_SERVER_DB_parametry"(DISCONNECT := #_w1,   // MB_SERVER
                           CONNECT_ID := 2,
                           IP_PORT := 503,
                           MB_HOLD_REG := "dbHold_RRG".Sending,
                           NDR => "CONFIG_MODBUS_TCP_SERVER"."CONFIG SERWER_2".ndr,
                           DR => "CONFIG_MODBUS_TCP_SERVER"."CONFIG SERWER_2".dr,
                           ERROR => "CONFIG_MODBUS_TCP_SERVER"."CONFIG SERWER_2".error,
                           STATUS => "CONFIG_MODBUS_TCP_SERVER"."CONFIG SERWER_2".STATUS);
END_REGION

REGION Network 5
   RUNG wire#powerrail
      I_Contact( "FirstScan" )
      Contact( "CONFIG_MODBUS_TCP_SERVER"."CONFIG SERWER_2".error )
      Move(in := "CONFIG_MODBUS_TCP_SERVER"."CONFIG SERWER_2".STATUS, out1 => "CONFIG_MODBUS_TCP_SERVER".ERROR_STATUS_SERWER_2)
   END_RUNG
   // the same network as SCL:
   IF NOT "FirstScan" AND "CONFIG_MODBUS_TCP_SERVER"."CONFIG SERWER_2".error THEN
       "CONFIG_MODBUS_TCP_SERVER".ERROR_STATUS_SERWER_2 := "CONFIG_MODBUS_TCP_SERVER"."CONFIG SERWER_2".STATUS;
   END_IF;
END_REGION

REGION Network 6: Czasy zadawane
   // Pobiera PLC 2 Zbiorniki
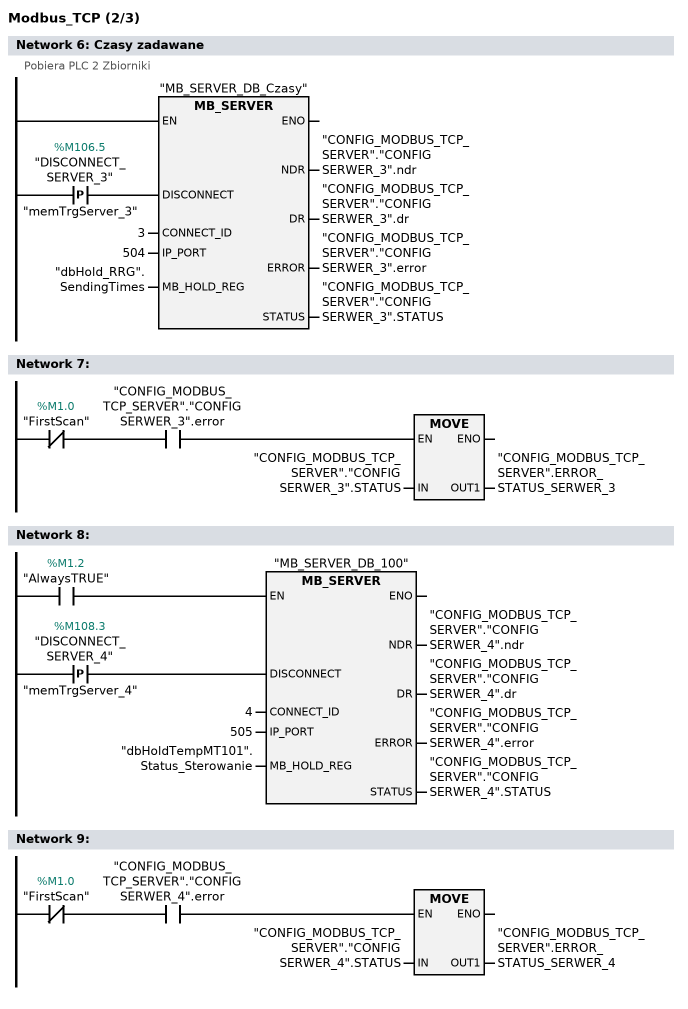
   RUNG wire#powerrail
      { S7_Templates := "[card1200 := 1, card1500 := 0]" } "MB_SERVER_DB_Czasy".MB_SERVER(DISCONNECT := wire#w1, CONNECT_ID := 3, IP_PORT := 504, MB_HOLD_REG := "dbHold_RRG".SendingTimes, NDR => "CONFIG_MODBUS_TCP_SERVER"."CONFIG SERWER_3".ndr, DR => "CONFIG_MODBUS_TCP_SERVER"."CONFIG SERWER_3".dr, ERROR => "CONFIG_MODBUS_TCP_SERVER"."CONFIG SERWER_3".error, STATUS => "CONFIG_MODBUS_TCP_SERVER"."CONFIG SERWER_3".STATUS)
   END_RUNG
   RUNG wire#powerrail
      P_Contact(operand := "DISCONNECT_SERVER_3", bit := "memTrgServer_3")
   END_RUNG wire#w1
   // the same network as SCL:
   #_w1 := "DISCONNECT_SERVER_3" AND NOT "memTrgServer_3";   // rising edge of "DISCONNECT_SERVER_3"
   "memTrgServer_3" := "DISCONNECT_SERVER_3";
   "MB_SERVER_DB_Czasy"(DISCONNECT := #_w1,   // MB_SERVER
                        CONNECT_ID := 3,
                        IP_PORT := 504,
                        MB_HOLD_REG := "dbHold_RRG".SendingTimes,
                        NDR => "CONFIG_MODBUS_TCP_SERVER"."CONFIG SERWER_3".ndr,
                        DR => "CONFIG_MODBUS_TCP_SERVER"."CONFIG SERWER_3".dr,
                        ERROR => "CONFIG_MODBUS_TCP_SERVER"."CONFIG SERWER_3".error,
                        STATUS => "CONFIG_MODBUS_TCP_SERVER"."CONFIG SERWER_3".STATUS);
END_REGION

REGION Network 7
   RUNG wire#powerrail
      I_Contact( "FirstScan" )
      Contact( "CONFIG_MODBUS_TCP_SERVER"."CONFIG SERWER_3".error )
      Move(in := "CONFIG_MODBUS_TCP_SERVER"."CONFIG SERWER_3".STATUS, out1 => "CONFIG_MODBUS_TCP_SERVER".ERROR_STATUS_SERWER_3)
   END_RUNG
   // the same network as SCL:
   IF NOT "FirstScan" AND "CONFIG_MODBUS_TCP_SERVER"."CONFIG SERWER_3".error THEN
       "CONFIG_MODBUS_TCP_SERVER".ERROR_STATUS_SERWER_3 := "CONFIG_MODBUS_TCP_SERVER"."CONFIG SERWER_3".STATUS;
   END_IF;
END_REGION

REGION Network 8
   RUNG wire#powerrail
      Contact( "AlwaysTRUE" )
      { S7_Templates := "[card1200 := 1, card1500 := 0]" } "MB_SERVER_DB_100".MB_SERVER(DISCONNECT := wire#w1, CONNECT_ID := 4, IP_PORT := 505, MB_HOLD_REG := "dbHoldTempMT101".Status_Sterowanie, NDR => "CONFIG_MODBUS_TCP_SERVER"."CONFIG SERWER_4".ndr, DR => "CONFIG_MODBUS_TCP_SERVER"."CONFIG SERWER_4".dr, ERROR => "CONFIG_MODBUS_TCP_SERVER"."CONFIG SERWER_4".error, STATUS => "CONFIG_MODBUS_TCP_SERVER"."CONFIG SERWER_4".STATUS)
   END_RUNG
   RUNG wire#powerrail
      P_Contact(operand := "DISCONNECT_SERVER_4", bit := "memTrgServer_4")
   END_RUNG wire#w1
   // the same network as SCL:
   #_w1 := "DISCONNECT_SERVER_4" AND NOT "memTrgServer_4";   // rising edge of "DISCONNECT_SERVER_4"
   "memTrgServer_4" := "DISCONNECT_SERVER_4";
   IF "AlwaysTRUE" THEN
       "MB_SERVER_DB_100"(DISCONNECT := #_w1,   // MB_SERVER
                          CONNECT_ID := 4,
                          IP_PORT := 505,
                          MB_HOLD_REG := "dbHoldTempMT101".Status_Sterowanie,
                          NDR => "CONFIG_MODBUS_TCP_SERVER"."CONFIG SERWER_4".ndr,
                          DR => "CONFIG_MODBUS_TCP_SERVER"."CONFIG SERWER_4".dr,
                          ERROR => "CONFIG_MODBUS_TCP_SERVER"."CONFIG SERWER_4".error,
                          STATUS => "CONFIG_MODBUS_TCP_SERVER"."CONFIG SERWER_4".STATUS);
   END_IF;
END_REGION

REGION Network 9
   RUNG wire#powerrail
      I_Contact( "FirstScan" )
      Contact( "CONFIG_MODBUS_TCP_SERVER"."CONFIG SERWER_4".error )
      Move(in := "CONFIG_MODBUS_TCP_SERVER"."CONFIG SERWER_4".STATUS, out1 => "CONFIG_MODBUS_TCP_SERVER".ERROR_STATUS_SERWER_4)
   END_RUNG
   // the same network as SCL:
   IF NOT "FirstScan" AND "CONFIG_MODBUS_TCP_SERVER"."CONFIG SERWER_4".error THEN
       "CONFIG_MODBUS_TCP_SERVER".ERROR_STATUS_SERWER_4 := "CONFIG_MODBUS_TCP_SERVER"."CONFIG SERWER_4".STATUS;
   END_IF;
END_REGION

REGION Network 10: Reakcja na błąd komunikacji
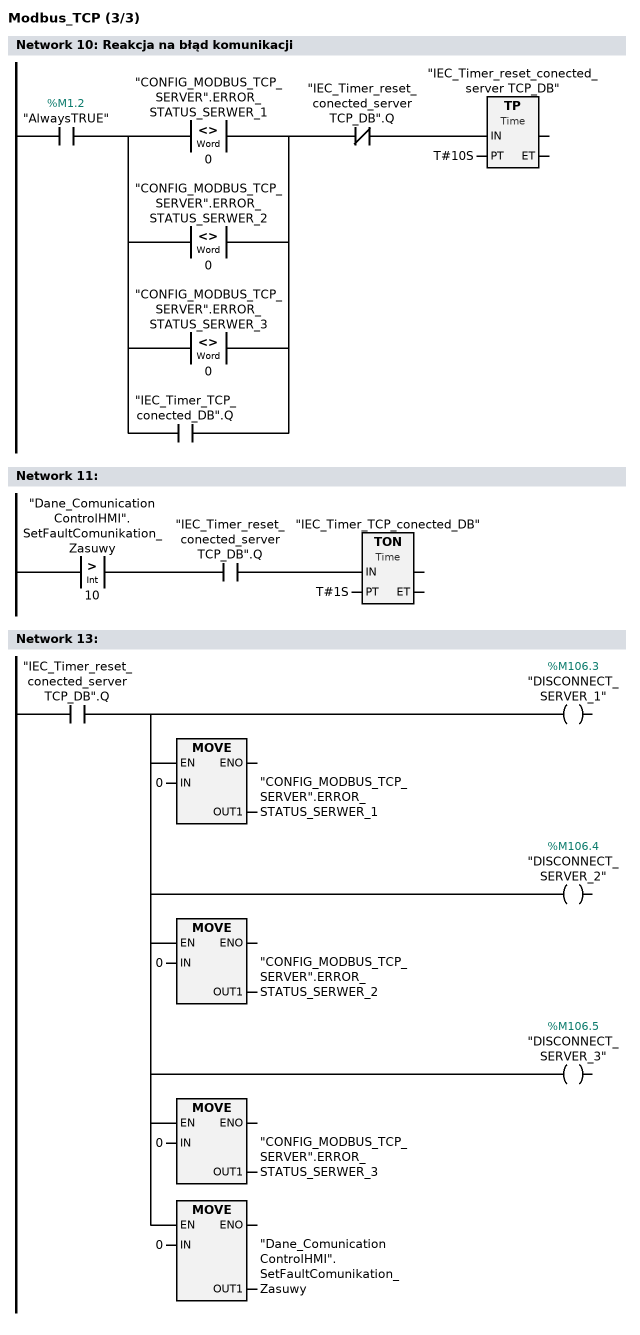
   RUNG wire#powerrail
      Contact( "AlwaysTRUE" )
      wire#w1
      { S7_Templates := "SrcType := Word" } NE_Contact(in1 := "CONFIG_MODBUS_TCP_SERVER".ERROR_STATUS_SERWER_1, in2 := 0)
      wire#w2
      I_Contact( "IEC_Timer_reset_conected_server TCP_DB".Q )
      { S7_Templates := "time_type := Time" } "IEC_Timer_reset_conected_server TCP_DB".TP(pt := T#10S, et =>)
   END_RUNG
   RUNG wire#w1
      { S7_Templates := "SrcType := Word" } NE_Contact(in1 := "CONFIG_MODBUS_TCP_SERVER".ERROR_STATUS_SERWER_2, in2 := 0)
   END_RUNG wire#w2
   RUNG wire#w1
      { S7_Templates := "SrcType := Word" } NE_Contact(in1 := "CONFIG_MODBUS_TCP_SERVER".ERROR_STATUS_SERWER_3, in2 := 0)
   END_RUNG wire#w2
   RUNG wire#w1
      Contact( "IEC_Timer_TCP_conected_DB".Q )
   END_RUNG wire#w2
   // the same network as SCL:
   "IEC_Timer_reset_conected_server TCP_DB".TP(IN := "AlwaysTRUE" AND (("CONFIG_MODBUS_TCP_SERVER".ERROR_STATUS_SERWER_1 <> 0) OR ("CONFIG_MODBUS_TCP_SERVER".ERROR_STATUS_SERWER_2 <> 0) OR ("CONFIG_MODBUS_TCP_SERVER".ERROR_STATUS_SERWER_3 <> 0) OR "IEC_Timer_TCP_conected_DB".Q) AND NOT "IEC_Timer_reset_conected_server TCP_DB".Q,
                           PT := T#10S);
END_REGION

REGION Network 11
   RUNG wire#powerrail
      { S7_Templates := "SrcType := Int" } GT_Contact(in1 := "Dane_ComunicationControlHMI".SetFaultComunikation_Zasuwy, in2 := 10)
      Contact( "IEC_Timer_reset_conected_server TCP_DB".Q )
      { S7_Templates := "time_type := Time" } "IEC_Timer_TCP_conected_DB".TON(pt := T#1S, et =>)
   END_RUNG
   // the same network as SCL:
   "IEC_Timer_TCP_conected_DB".TON(IN := ("Dane_ComunicationControlHMI".SetFaultComunikation_Zasuwy > 10) AND "IEC_Timer_reset_conected_server TCP_DB".Q,
                           PT := T#1S);
END_REGION

REGION Network 13
   RUNG wire#powerrail
      Contact( "IEC_Timer_reset_conected_server TCP_DB".Q )
      wire#w1
      Coil( "DISCONNECT_SERVER_1" )
   END_RUNG
   RUNG wire#w1
      Move(in := 0, out1 => "CONFIG_MODBUS_TCP_SERVER".ERROR_STATUS_SERWER_1)
   END_RUNG
   RUNG wire#w1
      Coil( "DISCONNECT_SERVER_2" )
   END_RUNG
   RUNG wire#w1
      Move(in := 0, out1 => "CONFIG_MODBUS_TCP_SERVER".ERROR_STATUS_SERWER_2)
   END_RUNG
   RUNG wire#w1
      Coil( "DISCONNECT_SERVER_3" )
   END_RUNG
   RUNG wire#w1
      Move(in := 0, out1 => "CONFIG_MODBUS_TCP_SERVER".ERROR_STATUS_SERWER_3)
   END_RUNG
   RUNG wire#w1
      Move(in := 0, out1 => "Dane_ComunicationControlHMI".SetFaultComunikation_Zasuwy)
   END_RUNG
   // the same network as SCL:
   "DISCONNECT_SERVER_1" := "IEC_Timer_reset_conected_server TCP_DB".Q;
   IF "IEC_Timer_reset_conected_server TCP_DB".Q THEN
       "CONFIG_MODBUS_TCP_SERVER".ERROR_STATUS_SERWER_1 := 0;
   END_IF;
   "DISCONNECT_SERVER_2" := "IEC_Timer_reset_conected_server TCP_DB".Q;
   IF "IEC_Timer_reset_conected_server TCP_DB".Q THEN
       "CONFIG_MODBUS_TCP_SERVER".ERROR_STATUS_SERWER_2 := 0;
   END_IF;
   "DISCONNECT_SERVER_3" := "IEC_Timer_reset_conected_server TCP_DB".Q;
   IF "IEC_Timer_reset_conected_server TCP_DB".Q THEN
       "CONFIG_MODBUS_TCP_SERVER".ERROR_STATUS_SERWER_3 := 0;
       "Dane_ComunicationControlHMI".SetFaultComunikation_Zasuwy := 0;
   END_IF;
END_REGION
END_FUNCTION_BLOCK

FUNCTION "IN" : Void
TITLE = Mapping control room inputs
{ S7_Optimized_Access := 'TRUE' }
AUTHOR : rtecmer
VERSION : 0.1
//Sprawdzanie wejść sterowniak i przekazanie sygnałów 

BEGIN
	(*
	Mapowanie wejść sterownika
	Sprawdzanie wejść sterowniak i przekazanie sygnałów 
	*)
	
	(*
	//=============================================================================
	//(JZWiK S.A Radosław Tecmer)
	//(c)Copyright (2021) All Rights Reserved
	//-----------------------------------------------------------------------------
	//Testowane z:   (system docelowy z  FW 4.4)
	//Pakiet inżynierski:   TIA Portal (V14 Sp1 Update 9)
	//Ograniczenia:  ( - )
	//Wymagania:  (minimalne S7-1200 CPU 1215C FW 4.2 .)
	//Funkcjonalnośc: (Mapowanie wejść sterownika
	//                 Sprawdzanie wejść sterowniak i przekazanie sygnałów )
	//-----------------------------------------------------------------------------
	//Zmainy wprowadzone:
	//Wersja  Data       Osoba wprowadzająca zmiany - ekspert
	//01.00.00 19.01.2022 (Tecmer Radosław - twórca) Pieresza wersja 01.00.00
	//=============================================================================
	*)
	
	// Pompy
	REGION Tryb sterowania Pompami
	  // ustawienie znacznika tryb pracy z systemu 1= Aut 0=REM
	  "inputRem_P1-P4" := "I2.4":P;
	  "IsRem" := "inputRem_P1-P4";
	  
	END_REGION
	
	// POMPA P1
	"IEC_Timer_P1_ready_DB".TOF(IN := "I0.1":P, // histereza na awarię
	                            PT := T#5S,
	                            Q => "inputReadyP1");
	                            
	
	
	"inputRunF_P1" :="I0.3":P;
	"inputRunS_P1" := "I0.2":P;
	
	// POMPA P2
	"IEC_Timer_P2_ready_DB".TOF(IN:="I0.5":P, // histereza na awarię
	                            PT:=T#5S,
	                            Q => "inputReadyP2" );
	
	
	"inputRunF_P2" := "I0.7":P;
	"inputRunS_P2" := "I0.6":P;
	
	// POMPA P3
	"IEC_Timer_P3_ready_DB".TOF(IN:="I1.1":P, // histereza na awarię
	                            PT:=T#5S,
	                            Q=>"inputReadyP3");
	
	
	"inputRunF_P3" := "I1.3":P;
	"inputRunS_P3" := "I1.2":P;
	
	// POMPA P4
	"IEC_Timer_P4_ready_DB".TOF(IN := "I1.5":P, // histereza na awarię
	                            PT := T#5S,
	                            Q => "inputReadyP4");
	
	
	"inputRunF_P4" := "I2.1":P;
	"inputRunS_P4" := "I2.0":P;
	
	
	// STOP AWARIA PRZYCISK
	"INPUTstopAccident_Pompy" := "I3.5":P;
	
	
	// ZASUWY Z11 Z12
	"inputREM_ZASUWY" := "I3.6":P;
	
	//Z12
	"imputRuchZ12":= "I3.1":P;
	"inputAwariaMomentZ12" := "I3.2":P;
	"inputOtwartaZ12" := "I3.3":P;
	"inputZamkniętaZ12" := "I3.4":P;
	"inputAumalokalneZ12" := "I4.4":P;
	"inputAumaautomatZ12" := "I4.5":P;
	"inputAumaawariaZ12" := "I4.6":P;
	"inputAumagotowośćZ12" := "I4.7":P;
	//Z11
	"inputRuchZ11" := "I2.5":P;
	"inputAwariaMomentZ11" := "I2.6":P;
	"inputOtwartaZ11" := "I2.7":P;
	"inputZamkniętaZ11" := "I3.0":P;
	"inputAumalokalneZ11" := "I4.0":P;
	"inputAumaautomatZ11" := "I4.1":P;
	"inputAumaawariaZ11" := "I4.2":P;
	"inputAumagotowośćZ11" := "I4.3":P;
	
	
	// ######################
	// Szafa RS Zasilanie OK
	"inputpowerOK_RS" := "I3.7":P;
	"Is_PowerRS5_OK" := "inputpowerOK_RS";
	// #########################
	
	// Gotowość P1
	REGION Gotowość P1
	  // Gdy brak sygnału na wejściu GOTO lub w statusie ustawiony bit awarii
	  // to brak gotowości
	  IF "inputReadyP1" = FALSE OR "bitH_Alarm_P1"= TRUE THEN
	    "IsReady_P1" := FALSE;
	  ELSE
	    "IsReady_P1" := TRUE;
	  END_IF;
	  
	END_REGION
	
	// Gotowość P2
	REGION Gotowość P2
	  // Gdy brak sygnału na wejściu GOTO lub w statusie ustawiony bit awarii
	  // to brak gotowości
	  IF "inputReadyP2" = FALSE OR "bitH_Alarm_P2" = TRUE THEN
	    "IsReady_P2" := FALSE;
	  ELSE
	    "IsReady_P2" := TRUE;
	  END_IF;
	  
	END_REGION
	
	// Gotowość P3
	REGION Gotowość P3
	  // Gdy brak sygnału na wejściu GOTO lub w statusie ustawiony bit awarii
	  // to brak gotowości
	  IF "inputReadyP3" = FALSE OR "bitH_Alarm_P3" = TRUE  THEN
	    "IsReady_P3" := FALSE;
	  ELSE
	    "IsReady_P3" := TRUE;
	  END_IF;
	  
	END_REGION
	
	// Gotowość P4
	REGION Gotowość P4
	  // Gdy brak sygnału na wejściu GOTO lub w statusie ustawiony bit awarii
	  // to brak gotowości
	  IF "inputReadyP4" = FALSE OR "bitH_Alarm_P4" = TRUE  THEN
	    "IsReady_P4" := FALSE;
	  ELSE
	    "IsReady_P4" := TRUE;
	  END_IF;
	  
	END_REGION
	
	
	
	
	// Gotowość falownika 
	"inputready_Inverter_P1-P4" := "I2.2":P;
	IF "inputready_Inverter_P1-P4" AND ("dbzarządzanie".awaria_falownika_F1 = False) THEN
	  // Ustaw gotowość
	  "IsReady_Inverter" :=TRUE;
	ELSE
	  "IsReady_Inverter" := FALSE;
	  ;
	END_IF;
	
	
	// Praca falownika 
	"inputrunInverter_" := "I2.3":P;
	"IsRunInverter1" := "inputrunInverter_";
	
	// potwierdzenie pracy Falownik Sieć
	// ***************
	//
	// ***************
	"IsRunInverter_P1" := "inputRunF_P1";
	"IsRunNetwork_P1" := "inputRunS_P1";
	"IsRunInverter_P2" := "inputRunF_P2";
	"IsRunNetwork_P2" := "inputRunS_P2";
	"IsRunInverter_P3" := "inputRunF_P3";
	"IsRunNetwork_P3" := "inputRunS_P3";
	"IsRunInverter_P4" := "inputRunF_P4";
	"IsRunNetwork_P4" := "inputRunS_P4";
	
	
	//************************
	//
	
	
	REGION Pompa P1
	  // Sygnał Run P1
	  IF "IsRunInverter_P1" OR "IsRunNetwork_P1" THEN
	    "IsRun_P1" := TRUE;
	  ELSE
	    "IsRun_P1" := FALSE;
	  END_IF;
	  
	END_REGION
	
	REGION Pompa P2
	  // Sygnał Run P2
	  IF "IsRunInverter_P2" OR "IsRunNetwork_P2" THEN
	    "IsRun_P2" := TRUE;
	  ELSE
	    "IsRun_P2" := FALSE;
	  END_IF;
	  
	END_REGION
	
	
	REGION Pompa P3
	  // Sygnał Run P3
	  IF "IsRunInverter_P3" OR "IsRunNetwork_P3" THEN
	    "IsRun_P3" := TRUE;
	  ELSE
	    "IsRun_P3" := FALSE;
	  END_IF;
	  
	END_REGION
	
	REGION Pompa P4
	  // Sygnał Run P4
	  IF "IsRunInverter_P4" OR "IsRunNetwork_P4" THEN
	    "IsRun_P4" := TRUE;
	  ELSE
	    "IsRun_P4" := FALSE;
	  END_IF;
	  
	END_REGION
	
	
	
	
	
	
	
	
END_FUNCTION

FUNCTION_BLOCK "filtr _kalmana_2"
{ S7_Optimized_Access := 'TRUE' }
VERSION : 0.1

BEGIN
	IF "FirstScan" THEN //w pierwszym cyklu sterownika
	  FOR "i(1)":= 0 TO 4 DO
	    "KALMAN_DB".kalman_K["i(1)"] := 0.0;
	    "KALMAN_DB".kalman_R["i(1)"] := 0.001;  //niepewność pomiaru
	    "KALMAN_DB".kalman_Q["i(1)"] := 0.00001;  //niepewność procesu
	    "KALMAN_DB".kalman_P["i(1)"] := 1.0;
	  END_FOR;        //parametry R i Q można dobrać osobno dla każdego kanału
	END_IF;           //zostaje wykonana inicjalizacja wszystkich 5 torów analogowych
	
	"R_TRIG_DB_CLK"(CLK:="Clock_10Hz", //oczekiwanie na zbocze narastające
	                Q => "zbocze_dod_zegar");
	                 
	                 
	IF "zbocze_dod_zegar" THEN  //ten fragment będzie wykonywany regularnie co 0.1s
	  
	  FOR "i(1)":= 0 TO 4 DO
	  
	    "KALMAN_DB".wejscie_anal["i(1)"] := PEEK_WORD(area:= 16#81, dbNumber:= 0, byteOffset:= (64 + (2 * "i(1)")));
	    //sterownik odczytuje kolejno pięć wejść analogowych,
	    //kazde z nich zajmuje w pamięci jedno słowo począwszy od adresu %IW64
	    
	    //"KALMAN_DB".wejscie_anal["I"] := "KALMAN_DB".wejscie_anal["I"] AND 16#03FF;
	    //maskowanie wejść
	  
	    "KALMAN_DB".pomiar_napiecie["i(1)"] := NORM_X(MIN:= 0, VALUE:= "KALMAN_DB".wejscie_anal["i(1)"], MAX:= 27648);
	    //wartość zwracana przez n-bitowy przetwornik A\C zawiera się w przedziale od 0 do (2^n)-1
	  
	    "KALMAN_DB".pomiar_napiecie["i(1)"] := "KALMAN_DB".pomiar_napiecie["i(1)"] * 10.0;
	    //znormalizowana wartość zostaje pomnożona przez 10.0, aby tagi w tablicy "pomiar_napiecie"
	    //reprezentowały faktyczne napięcie na wejściu analogowym
	    //w przypadku zakresów wejściowych różnych od standardu można
	    //skorzystać z intruksji CASE i mnożyć wyjście przez różne skalary
	  
	    //FILTR KALMANA
	    "KALMAN_DB".kalman_P["i(1)"] := "KALMAN_DB".kalman_P["i(1)"] + "KALMAN_DB".kalman_Q["i(1)"]; //predykcja
	  
	    "KALMAN_DB".kalman_K["i(1)"] := "KALMAN_DB".kalman_P["i(1)"] / ("KALMAN_DB".kalman_P["i(1)"] + "KALMAN_DB".kalman_R["i(1)"]); //korekcja
	    
	    "KALMAN_DB".kalman_napiecie["i(1)"] := "KALMAN_DB".kalman_napiecie["i(1)"] +
	    "KALMAN_DB".kalman_K["i(1)"] * ("KALMAN_DB".pomiar_napiecie["i(1)"] - "KALMAN_DB".kalman_napiecie["i(1)"]);
	    
	    "KALMAN_DB".kalman_P["i(1)"] := (1.0 - "KALMAN_DB".kalman_K["i(1)"]) * "KALMAN_DB".kalman_P["i(1)"];
	  
	    //wynik filtracji gotowy do użycia znajduje się w tablicy "KALMAN_DB".kalman_napiecie
	  
	  END_FOR;
	  
	END_IF;
	
END_FUNCTION_BLOCK

FUNCTION_BLOCK "Byte status zasuw"
TITLE = Calculation Byte Status M1-M4
{ S7_Optimized_Access := 'TRUE' }
AUTHOR : rtecmer
VERSION : 0.1
//Byte określający ile napędów dostępnych. Wykorzystywany do blokowania przełączenia na sieć ostatniej dostępnej pompy.

BEGIN
	(*
	//=============================================================================
	//(JZWiK S.A Radosław Tecmer)
	//(c)Copyright (2021) All Rights Reserved
	//-----------------------------------------------------------------------------
	//Testowane z:   (system docelowy z  FW 4.4)
	//Pakiet inżynierski:   TIA Portal (V14 Sp1 Update 9)
	//Ograniczenia:  ( - )
	//Wymagania:  (minimalne S7-1200 CPU 1215C FW 4.2 .)
	//Funkcjonalnośc: (Byte statusu napędów Z11 Z12 Zasuwy )
	//-----------------------------------------------------------------------------
	//Zmainy wprowadzone:
	//Wersja  Data       Osoba wprowadzająca zmiany - ekspert
	//01.00.00 17.11.2021 (Tecmer Radosław - twórca) Pieresza wersja 01.00.00
	//=============================================================================
	*)
	
	
	
	
	
	REGION przekazanie satusu Z11 Z12  do znacznika
	  //przekazanie
	  // Z11 Przekazanie Byte H ststusu do Byte znacznika 
	  "Byte_Status_Z11" := %DB100.DBB29;
	  // Z12 Przekazanie Byte H ststusu do Byte znacznika 
	  "Byte_Status_Z12" := %DB100.DBB31;
	
	  
	  
	END_REGION
	
END_FUNCTION_BLOCK

FUNCTION_BLOCK "FB220_TimeSyn_PLC_To_HMI"
{ S7_Optimized_Access := 'FALSE' }
VERSION : 0.1
   VAR_OUTPUT 
      PLC_RD_LOC_T {InstructionName := 'DTL'; LibVersion := '1.0'} : DTL;
      PLC_RD_SYS_T {InstructionName := 'DTL'; LibVersion := '1.0'} : DTL;
   END_VAR

   VAR_IN_OUT 
      AreaPointer_JobMailbox : Array[0..3] of Word;
      SetTime : Bool;
      SetDate : Bool;
   END_VAR

   VAR 
      Func_RD_LOC_T {InstructionName := 'DTL'; LibVersion := '1.0'} : DTL;
      Ret_Val_RD_LOC_T : Int;
      BCD_Hour : Word;
      BCD_Minute : Word;
      BCD_Second : Word;
      BCD_Weekdday : Word;
      BCD_Day : Word;
      BCD_Month : Word;
      BCD32_Year : DWord;
      BCD16_Year : Word;
      STEP1 : Bool;
      STEP2 : Bool;
      STEP3 : Bool;
      STEP10 : Bool;
      STEP11 : Bool;
      STEP12 : Bool;
      Func_RD_SYS_T {InstructionName := 'DTL'; LibVersion := '1.0'} : DTL;
      Ret_Val_RD_SYS_T : Int;
   END_VAR


BEGIN
	//SIMATIC S7-1200 / 1500
	//
	
	//Odczyt aktualnego czasu PLC // Odczyt aktualnego czasu PLC
	#Ret_Val_RD_LOC_T := RD_LOC_T(#Func_RD_LOC_T);
	#PLC_RD_LOC_T := (#Func_RD_LOC_T);
	#Ret_Val_RD_SYS_T := RD_SYS_T(#Func_RD_SYS_T);
	#PLC_RD_SYS_T := (#Func_RD_SYS_T);
	
	
	//***Czas transmisja
	//Step 1
	//Zacznij, jeśli job mailmox  ma wartość zero.    
	IF #SetTime AND (#AreaPointer_JobMailbox[0] = 0) THEN
	    
	    //Parameter 1-3: Mit Null "0" vorbelegen //Parameters 1-3: Preassign with zero "0"
	    #AreaPointer_JobMailbox[1] := 0;
	    #AreaPointer_JobMailbox[2] := 0;
	    #AreaPointer_JobMailbox[3] := 0;
	    
	    #SetTime := false;
	    #STEP2 := true;
	    
	END_IF;
	
	//Step 2
	//plc job 14 - assign parameter
	IF #STEP2 THEN
	    
	    //Convert USInt to BCD format (plc job 14 need bcd format)
	    #BCD_Hour := INT_TO_BCD16(#Func_RD_LOC_T.HOUR);
	    #BCD_Minute := INT_TO_BCD16(#Func_RD_LOC_T.MINUTE);
	    #BCD_Second := INT_TO_BCD16(#Func_RD_LOC_T.SECOND);
	    
	    //Parameter
	    #AreaPointer_JobMailbox[1].%B0 := #BCD_Hour.%B0;
	    #AreaPointer_JobMailbox[2].%B1 := #BCD_Minute.%B0;
	    #AreaPointer_JobMailbox[2].%B0 := #BCD_Second.%B0;
	    
	    //plc job 14
	    #AreaPointer_JobMailbox[0] := 14;
	    
	    #STEP2 := FALSE;
	    
	END_IF;
	
	
	//****Data przesłania
	//Step 10
	//Start, if job mailbox are zero.    
	IF #SetDate AND (#AreaPointer_JobMailbox[0] = 0) THEN
	    
	    //Parameters 1-3: Preassign with zero "0"
	    #AreaPointer_JobMailbox[1] := 0;
	    #AreaPointer_JobMailbox[2] := 0;
	    #AreaPointer_JobMailbox[3] := 0;
	    
	    #SetDate := false;
	    #STEP11 := true;
	    
	END_IF;
	
